// TwinCAT 3 PLC project TcoIoBeckhoff
// Title: TcoIoBeckhoff
// Company: Vortex.Library
// ProjectVersion: 1.19.1.1780
// ProgramVersion: 3.1.4023.0
// libraries:
//   Tc2_EtherCAT, * (Beckhoff Automation GmbH)
//   Tc2_Standard, * (Beckhoff Automation GmbH)
//   Tc2_System, * (Beckhoff Automation GmbH)
//   Tc3_Module, * (Beckhoff Automation GmbH)
//   TcoCore, 1.19.1.1780 (Vortex.Library)
// project tree:
//   Diagnostics/EtherCAT/MasterDevice/ InfoData_E68C61CD.TcDUT (not stored), Inputs_A65FACA4.TcDUT (not stored), Outputs_23C0ED1D.TcDUT (not stored), TcoEthercatDiagnosticsTask.TcPOU, TcoEthercatMasterDeviceState.TcDUT (not stored), ITcoEthercatMasterDevice.TcIO (not stored), TcoEthercatMasterDevice.TcPOU
//   Diagnostics/EtherCAT/MasterDevice/Messenger/ DiagnosticsMessenger.TcPOU (not stored), DiagnosticsMessengers.TcPOU (not stored)
//   Diagnostics/EtherCAT/SyncUnit/ SyncUnitTask_2D604ED5.TcDUT (not stored), TcoSyncUnit.TcPOU, InfoData_2A97D6CF.TcDUT (not stored), ITcoSyncUnit.TcIO (not stored), SyncUnitState.TcDUT (not stored), WcState_0B2B16F9.TcDUT (not stored)
//   Diagnostics/EtherCAT/ TcoEthercat.TcGVL (not stored)
//   / PlcTask.TcTTO (not stored)
//   POUs/ MAIN.TcPOU
// real-time tasks:
//   TASK PlcTask: cycle T#10ms, priority 20, ADS port 350
//   TASK PlcTask1: cycle T#10ms, priority 21, ADS port 351
//   TASK PlcTask2: cycle T#10ms, priority 22, ADS port 352
// I/O:
//   DEVICE Device 1 (EtherCAT), AmsNetId 172.20.10.104.2.1
//     Term 1 (EK1200) [EK1200-5000 EtherCAT Power supply (2A E-Bus)]
//       Term 2 (EL6002) [EL6002 Interface 2Ch. (RS232)]
//       Term 3 (EL1809) [EL1809 16Ch. Dig. Input 24V, 3ms]
//       Term 4 (EL2809) [EL2809 16Ch. Dig. Output 24V, 0.5A]
//       Term 5 (EL4004) [EL4004 4Ch. Ana. Output 0-10V, 12bit]
//       Term 6 (EL2809) [EL2809 16Ch. Dig. Output 24V, 0.5A]
//       Term 7 (EL6001) [EL6001 Interface (RS232)]
//       Term 8 (EL9011) [EL9011 End Terminal]
//   DEVICE Device 4 (EtherCAT), AmsNetId 172.20.10.104.5.1
//     Term 9 (EK1100) [EK1100 EtherCAT Coupler (2A E-Bus)]
//       Term 10 (EL6001) [EL6001 Interface (RS232)]
//       Term 11 (EL1809) [EL1809 16Ch. Dig. Input 24V, 3ms]
//       Term 12 (EL2809) [EL2809 16Ch. Dig. Output 24V, 0.5A]
//       Term 13 (EK1110) [EK1110 EtherCAT extension]
//     Term 14 (EK1100) [EK1100 EtherCAT Coupler (2A E-Bus)]
//       Term 15 (EL3403) [EL3403 3Ch. Power Measuring]
//       Term 16 (EK1122) [EK1122 2 port EtherCAT junction]
//         Term 17 (EK1100) [EK1100 EtherCAT Coupler (2A E-Bus)]
//           Term 18 (EL3174-0002) [EL3174-0002 4Ch. Ana. Input +/-10V, +/-20mA 16 Bit, Isolated Channels]
//           Term 19 (EL6001) [EL6001 Interface (RS232)]
//           Term 20 (EL3011) [EL3011 4Ch. Ana. Input 0-20mA DIFF]
//           Term 21 (EL2008) [EL2008 8Ch. Dig. Output 24V, 0.5A]
//           Term 22 (EL2008) [EL2008 8Ch. Dig. Output 24V, 0.5A]
//           Term 16 (EL9011) [EL9011 End Terminal]
//       Term 23 (EL3024) [EL3024 4Ch. Ana. Input 4-20mA DIFF]
//       Term 17 (EL9011) [EL9011 End Terminal]
// variable links:
//   TcoIoBeckhoffTests/TcoIoBeckhoffTests Instance <-> Device 1 (EtherCAT)
//     PlcTask Inputs/GVL_iXlinker.Device_1_EtherCAT.InfoData.AmsNetId <-> InfoData/AmsNetId
//     PlcTask Inputs/GVL_iXlinker.Device_1_EtherCAT.InfoData.CfgSlaveCount <-> InfoData/CfgSlaveCount
//     PlcTask Inputs/GVL_iXlinker.Device_1_EtherCAT.InfoData.ChangeCount <-> InfoData/ChangeCount
//     PlcTask Inputs/GVL_iXlinker.Device_1_EtherCAT.InfoData.DcToExtTimeOffset <-> InfoData/DcToExtTimeOffset
//     PlcTask Inputs/GVL_iXlinker.Device_1_EtherCAT.InfoData.DcToTcTimeOffset <-> InfoData/DcToTcTimeOffset
//     PlcTask Inputs/GVL_iXlinker.Device_1_EtherCAT.InfoData.DevId <-> InfoData/DevId
//     PlcTask Inputs/GVL_iXlinker.Device_1_EtherCAT.Inputs.DevState <-> Inputs/DevState
//     PlcTask Inputs/GVL_iXlinker.Device_1_EtherCAT.Inputs.Frm0InputToggle <-> Inputs/Frm0InputToggle
//     PlcTask Inputs/GVL_iXlinker.Device_1_EtherCAT.Inputs.Frm0State <-> Inputs/Frm0State
//     PlcTask Inputs/GVL_iXlinker.Device_1_EtherCAT.Inputs.Frm0WcState <-> Inputs/Frm0WcState
//     PlcTask Inputs/GVL_iXlinker.Device_1_EtherCAT.Inputs.SlaveCount <-> Inputs/SlaveCount
//     PlcTask Inputs/GVL_iXlinker.Device_1_EtherCAT.SyncUnits._default.PlcTask1.InfoData.ObjectId <-> SyncUnits/<default>/PlcTask1/InfoData/ObjectId
//     PlcTask Inputs/GVL_iXlinker.Device_1_EtherCAT.SyncUnits._default.PlcTask1.InfoData.SlaveCount <-> SyncUnits/<default>/PlcTask1/InfoData/SlaveCount
//     PlcTask Inputs/GVL_iXlinker.Device_1_EtherCAT.SyncUnits._default.PlcTask1.InfoData.State <-> SyncUnits/<default>/PlcTask1/InfoData/State
//     PlcTask Inputs/GVL_iXlinker.Device_1_EtherCAT.SyncUnits._default.PlcTask1.WcState.WcState <-> SyncUnits/<default>/PlcTask1/WcState/WcState
//     PlcTask Outputs/GVL_iXlinker.Device_1_EtherCAT.Outputs.DevCtrl <-> Outputs/DevCtrl
//     PlcTask Outputs/GVL_iXlinker.Device_1_EtherCAT.Outputs.Frm0Ctrl <-> Outputs/Frm0Ctrl
//     PlcTask Outputs/GVL_iXlinker.Device_1_EtherCAT.Outputs.Frm0WcCtrl <-> Outputs/Frm0WcCtrl
//   TcoIoBeckhoffTests/TcoIoBeckhoffTests Instance <-> Device 1 (EtherCAT)/Term 1 (EK1200)/Term 2 (EL6002)
//     PlcTask Inputs/GVL_iXlinker.Device_1_EtherCAT.Term_1_EK1200.Term_2_EL6002.COM_TxPDO_Map_Inputs_Channel_1.Data_In[0] <-> COM TxPDO-Map Inputs Channel 1/Data In 0
//     PlcTask Inputs/GVL_iXlinker.Device_1_EtherCAT.Term_1_EK1200.Term_2_EL6002.COM_TxPDO_Map_Inputs_Channel_1.Data_In[10] <-> COM TxPDO-Map Inputs Channel 1/Data In 10
//     PlcTask Inputs/GVL_iXlinker.Device_1_EtherCAT.Term_1_EK1200.Term_2_EL6002.COM_TxPDO_Map_Inputs_Channel_1.Data_In[11] <-> COM TxPDO-Map Inputs Channel 1/Data In 11
//     PlcTask Inputs/GVL_iXlinker.Device_1_EtherCAT.Term_1_EK1200.Term_2_EL6002.COM_TxPDO_Map_Inputs_Channel_1.Data_In[12] <-> COM TxPDO-Map Inputs Channel 1/Data In 12
//     PlcTask Inputs/GVL_iXlinker.Device_1_EtherCAT.Term_1_EK1200.Term_2_EL6002.COM_TxPDO_Map_Inputs_Channel_1.Data_In[13] <-> COM TxPDO-Map Inputs Channel 1/Data In 13
//     PlcTask Inputs/GVL_iXlinker.Device_1_EtherCAT.Term_1_EK1200.Term_2_EL6002.COM_TxPDO_Map_Inputs_Channel_1.Data_In[14] <-> COM TxPDO-Map Inputs Channel 1/Data In 14
//     PlcTask Inputs/GVL_iXlinker.Device_1_EtherCAT.Term_1_EK1200.Term_2_EL6002.COM_TxPDO_Map_Inputs_Channel_1.Data_In[15] <-> COM TxPDO-Map Inputs Channel 1/Data In 15
//     PlcTask Inputs/GVL_iXlinker.Device_1_EtherCAT.Term_1_EK1200.Term_2_EL6002.COM_TxPDO_Map_Inputs_Channel_1.Data_In[16] <-> COM TxPDO-Map Inputs Channel 1/Data In 16
//     PlcTask Inputs/GVL_iXlinker.Device_1_EtherCAT.Term_1_EK1200.Term_2_EL6002.COM_TxPDO_Map_Inputs_Channel_1.Data_In[17] <-> COM TxPDO-Map Inputs Channel 1/Data In 17
//     PlcTask Inputs/GVL_iXlinker.Device_1_EtherCAT.Term_1_EK1200.Term_2_EL6002.COM_TxPDO_Map_Inputs_Channel_1.Data_In[18] <-> COM TxPDO-Map Inputs Channel 1/Data In 18
//     PlcTask Inputs/GVL_iXlinker.Device_1_EtherCAT.Term_1_EK1200.Term_2_EL6002.COM_TxPDO_Map_Inputs_Channel_1.Data_In[19] <-> COM TxPDO-Map Inputs Channel 1/Data In 19
//     PlcTask Inputs/GVL_iXlinker.Device_1_EtherCAT.Term_1_EK1200.Term_2_EL6002.COM_TxPDO_Map_Inputs_Channel_1.Data_In[1] <-> COM TxPDO-Map Inputs Channel 1/Data In 1
//     PlcTask Inputs/GVL_iXlinker.Device_1_EtherCAT.Term_1_EK1200.Term_2_EL6002.COM_TxPDO_Map_Inputs_Channel_1.Data_In[20] <-> COM TxPDO-Map Inputs Channel 1/Data In 20
//     PlcTask Inputs/GVL_iXlinker.Device_1_EtherCAT.Term_1_EK1200.Term_2_EL6002.COM_TxPDO_Map_Inputs_Channel_1.Data_In[21] <-> COM TxPDO-Map Inputs Channel 1/Data In 21
//     PlcTask Inputs/GVL_iXlinker.Device_1_EtherCAT.Term_1_EK1200.Term_2_EL6002.COM_TxPDO_Map_Inputs_Channel_1.Data_In[2] <-> COM TxPDO-Map Inputs Channel 1/Data In 2
//     PlcTask Inputs/GVL_iXlinker.Device_1_EtherCAT.Term_1_EK1200.Term_2_EL6002.COM_TxPDO_Map_Inputs_Channel_1.Data_In[3] <-> COM TxPDO-Map Inputs Channel 1/Data In 3
//     PlcTask Inputs/GVL_iXlinker.Device_1_EtherCAT.Term_1_EK1200.Term_2_EL6002.COM_TxPDO_Map_Inputs_Channel_1.Data_In[4] <-> COM TxPDO-Map Inputs Channel 1/Data In 4
//     PlcTask Inputs/GVL_iXlinker.Device_1_EtherCAT.Term_1_EK1200.Term_2_EL6002.COM_TxPDO_Map_Inputs_Channel_1.Data_In[5] <-> COM TxPDO-Map Inputs Channel 1/Data In 5
//     PlcTask Inputs/GVL_iXlinker.Device_1_EtherCAT.Term_1_EK1200.Term_2_EL6002.COM_TxPDO_Map_Inputs_Channel_1.Data_In[6] <-> COM TxPDO-Map Inputs Channel 1/Data In 6
//     PlcTask Inputs/GVL_iXlinker.Device_1_EtherCAT.Term_1_EK1200.Term_2_EL6002.COM_TxPDO_Map_Inputs_Channel_1.Data_In[7] <-> COM TxPDO-Map Inputs Channel 1/Data In 7
//     PlcTask Inputs/GVL_iXlinker.Device_1_EtherCAT.Term_1_EK1200.Term_2_EL6002.COM_TxPDO_Map_Inputs_Channel_1.Data_In[8] <-> COM TxPDO-Map Inputs Channel 1/Data In 8
//     PlcTask Inputs/GVL_iXlinker.Device_1_EtherCAT.Term_1_EK1200.Term_2_EL6002.COM_TxPDO_Map_Inputs_Channel_1.Data_In[9] <-> COM TxPDO-Map Inputs Channel 1/Data In 9
//     PlcTask Inputs/GVL_iXlinker.Device_1_EtherCAT.Term_1_EK1200.Term_2_EL6002.COM_TxPDO_Map_Inputs_Channel_2.Data_In[0] <-> COM TxPDO-Map Inputs Channel 2/Data In 0
//     PlcTask Inputs/GVL_iXlinker.Device_1_EtherCAT.Term_1_EK1200.Term_2_EL6002.COM_TxPDO_Map_Inputs_Channel_2.Data_In[10] <-> COM TxPDO-Map Inputs Channel 2/Data In 10
//     PlcTask Inputs/GVL_iXlinker.Device_1_EtherCAT.Term_1_EK1200.Term_2_EL6002.COM_TxPDO_Map_Inputs_Channel_2.Data_In[11] <-> COM TxPDO-Map Inputs Channel 2/Data In 11
//     PlcTask Inputs/GVL_iXlinker.Device_1_EtherCAT.Term_1_EK1200.Term_2_EL6002.COM_TxPDO_Map_Inputs_Channel_2.Data_In[12] <-> COM TxPDO-Map Inputs Channel 2/Data In 12
//     PlcTask Inputs/GVL_iXlinker.Device_1_EtherCAT.Term_1_EK1200.Term_2_EL6002.COM_TxPDO_Map_Inputs_Channel_2.Data_In[13] <-> COM TxPDO-Map Inputs Channel 2/Data In 13
//     PlcTask Inputs/GVL_iXlinker.Device_1_EtherCAT.Term_1_EK1200.Term_2_EL6002.COM_TxPDO_Map_Inputs_Channel_2.Data_In[14] <-> COM TxPDO-Map Inputs Channel 2/Data In 14
//     PlcTask Inputs/GVL_iXlinker.Device_1_EtherCAT.Term_1_EK1200.Term_2_EL6002.COM_TxPDO_Map_Inputs_Channel_2.Data_In[15] <-> COM TxPDO-Map Inputs Channel 2/Data In 15
//     PlcTask Inputs/GVL_iXlinker.Device_1_EtherCAT.Term_1_EK1200.Term_2_EL6002.COM_TxPDO_Map_Inputs_Channel_2.Data_In[16] <-> COM TxPDO-Map Inputs Channel 2/Data In 16
//     PlcTask Inputs/GVL_iXlinker.Device_1_EtherCAT.Term_1_EK1200.Term_2_EL6002.COM_TxPDO_Map_Inputs_Channel_2.Data_In[17] <-> COM TxPDO-Map Inputs Channel 2/Data In 17
//     PlcTask Inputs/GVL_iXlinker.Device_1_EtherCAT.Term_1_EK1200.Term_2_EL6002.COM_TxPDO_Map_Inputs_Channel_2.Data_In[18] <-> COM TxPDO-Map Inputs Channel 2/Data In 18
//     PlcTask Inputs/GVL_iXlinker.Device_1_EtherCAT.Term_1_EK1200.Term_2_EL6002.COM_TxPDO_Map_Inputs_Channel_2.Data_In[19] <-> COM TxPDO-Map Inputs Channel 2/Data In 19
//     PlcTask Inputs/GVL_iXlinker.Device_1_EtherCAT.Term_1_EK1200.Term_2_EL6002.COM_TxPDO_Map_Inputs_Channel_2.Data_In[1] <-> COM TxPDO-Map Inputs Channel 2/Data In 1
//     PlcTask Inputs/GVL_iXlinker.Device_1_EtherCAT.Term_1_EK1200.Term_2_EL6002.COM_TxPDO_Map_Inputs_Channel_2.Data_In[20] <-> COM TxPDO-Map Inputs Channel 2/Data In 20
//     PlcTask Inputs/GVL_iXlinker.Device_1_EtherCAT.Term_1_EK1200.Term_2_EL6002.COM_TxPDO_Map_Inputs_Channel_2.Data_In[21] <-> COM TxPDO-Map Inputs Channel 2/Data In 21
//     PlcTask Inputs/GVL_iXlinker.Device_1_EtherCAT.Term_1_EK1200.Term_2_EL6002.COM_TxPDO_Map_Inputs_Channel_2.Data_In[2] <-> COM TxPDO-Map Inputs Channel 2/Data In 2
//     PlcTask Inputs/GVL_iXlinker.Device_1_EtherCAT.Term_1_EK1200.Term_2_EL6002.COM_TxPDO_Map_Inputs_Channel_2.Data_In[3] <-> COM TxPDO-Map Inputs Channel 2/Data In 3
//     PlcTask Inputs/GVL_iXlinker.Device_1_EtherCAT.Term_1_EK1200.Term_2_EL6002.COM_TxPDO_Map_Inputs_Channel_2.Data_In[4] <-> COM TxPDO-Map Inputs Channel 2/Data In 4
//     PlcTask Inputs/GVL_iXlinker.Device_1_EtherCAT.Term_1_EK1200.Term_2_EL6002.COM_TxPDO_Map_Inputs_Channel_2.Data_In[5] <-> COM TxPDO-Map Inputs Channel 2/Data In 5
//     PlcTask Inputs/GVL_iXlinker.Device_1_EtherCAT.Term_1_EK1200.Term_2_EL6002.COM_TxPDO_Map_Inputs_Channel_2.Data_In[6] <-> COM TxPDO-Map Inputs Channel 2/Data In 6
//     PlcTask Inputs/GVL_iXlinker.Device_1_EtherCAT.Term_1_EK1200.Term_2_EL6002.COM_TxPDO_Map_Inputs_Channel_2.Data_In[7] <-> COM TxPDO-Map Inputs Channel 2/Data In 7
//     PlcTask Inputs/GVL_iXlinker.Device_1_EtherCAT.Term_1_EK1200.Term_2_EL6002.COM_TxPDO_Map_Inputs_Channel_2.Data_In[8] <-> COM TxPDO-Map Inputs Channel 2/Data In 8
//     PlcTask Inputs/GVL_iXlinker.Device_1_EtherCAT.Term_1_EK1200.Term_2_EL6002.COM_TxPDO_Map_Inputs_Channel_2.Data_In[9] <-> COM TxPDO-Map Inputs Channel 2/Data In 9
//     PlcTask Inputs/GVL_iXlinker.Device_1_EtherCAT.Term_1_EK1200.Term_2_EL6002.COM_TxPDO_Map_Inputs_Channel_1.Status/Buffer_full <-> COM TxPDO-Map Inputs Channel 1/Status/Buffer full
//     PlcTask Inputs/GVL_iXlinker.Device_1_EtherCAT.Term_1_EK1200.Term_2_EL6002.COM_TxPDO_Map_Inputs_Channel_2.Status/Buffer_full <-> COM TxPDO-Map Inputs Channel 2/Status/Buffer full
//     PlcTask Inputs/GVL_iXlinker.Device_1_EtherCAT.Term_1_EK1200.Term_2_EL6002.COM_TxPDO_Map_Inputs_Channel_1.Status/Framing_error <-> COM TxPDO-Map Inputs Channel 1/Status/Framing error
//     PlcTask Inputs/GVL_iXlinker.Device_1_EtherCAT.Term_1_EK1200.Term_2_EL6002.COM_TxPDO_Map_Inputs_Channel_2.Status/Framing_error <-> COM TxPDO-Map Inputs Channel 2/Status/Framing error
//     PlcTask Inputs/GVL_iXlinker.Device_1_EtherCAT.Term_1_EK1200.Term_2_EL6002.COM_TxPDO_Map_Inputs_Channel_1.Status/Init_accepted <-> COM TxPDO-Map Inputs Channel 1/Status/Init accepted
//     PlcTask Inputs/GVL_iXlinker.Device_1_EtherCAT.Term_1_EK1200.Term_2_EL6002.COM_TxPDO_Map_Inputs_Channel_2.Status/Init_accepted <-> COM TxPDO-Map Inputs Channel 2/Status/Init accepted
//     PlcTask Inputs/GVL_iXlinker.Device_1_EtherCAT.Term_1_EK1200.Term_2_EL6002.COM_TxPDO_Map_Inputs_Channel_1.Status/Input_length <-> COM TxPDO-Map Inputs Channel 1/Status/Input length
//     PlcTask Inputs/GVL_iXlinker.Device_1_EtherCAT.Term_1_EK1200.Term_2_EL6002.COM_TxPDO_Map_Inputs_Channel_2.Status/Input_length <-> COM TxPDO-Map Inputs Channel 2/Status/Input length
//     PlcTask Inputs/GVL_iXlinker.Device_1_EtherCAT.Term_1_EK1200.Term_2_EL6002.COM_TxPDO_Map_Inputs_Channel_1.Status/Overrun_error <-> COM TxPDO-Map Inputs Channel 1/Status/Overrun error
//     PlcTask Inputs/GVL_iXlinker.Device_1_EtherCAT.Term_1_EK1200.Term_2_EL6002.COM_TxPDO_Map_Inputs_Channel_2.Status/Overrun_error <-> COM TxPDO-Map Inputs Channel 2/Status/Overrun error
//     PlcTask Inputs/GVL_iXlinker.Device_1_EtherCAT.Term_1_EK1200.Term_2_EL6002.COM_TxPDO_Map_Inputs_Channel_1.Status/Parity_error <-> COM TxPDO-Map Inputs Channel 1/Status/Parity error
//     PlcTask Inputs/GVL_iXlinker.Device_1_EtherCAT.Term_1_EK1200.Term_2_EL6002.COM_TxPDO_Map_Inputs_Channel_2.Status/Parity_error <-> COM TxPDO-Map Inputs Channel 2/Status/Parity error
//     PlcTask Inputs/GVL_iXlinker.Device_1_EtherCAT.Term_1_EK1200.Term_2_EL6002.COM_TxPDO_Map_Inputs_Channel_1.Status/Receive_request <-> COM TxPDO-Map Inputs Channel 1/Status/Receive request
//     PlcTask Inputs/GVL_iXlinker.Device_1_EtherCAT.Term_1_EK1200.Term_2_EL6002.COM_TxPDO_Map_Inputs_Channel_2.Status/Receive_request <-> COM TxPDO-Map Inputs Channel 2/Status/Receive request
//     PlcTask Inputs/GVL_iXlinker.Device_1_EtherCAT.Term_1_EK1200.Term_2_EL6002.COM_TxPDO_Map_Inputs_Channel_1.Status/Transmit_accepted <-> COM TxPDO-Map Inputs Channel 1/Status/Transmit accepted
//     PlcTask Inputs/GVL_iXlinker.Device_1_EtherCAT.Term_1_EK1200.Term_2_EL6002.COM_TxPDO_Map_Inputs_Channel_2.Status/Transmit_accepted <-> COM TxPDO-Map Inputs Channel 2/Status/Transmit accepted
//     PlcTask Inputs/GVL_iXlinker.Device_1_EtherCAT.Term_1_EK1200.Term_2_EL6002.InfoData.AdsAddr <-> InfoData/AdsAddr
//     PlcTask Inputs/GVL_iXlinker.Device_1_EtherCAT.Term_1_EK1200.Term_2_EL6002.InfoData.ObjectId <-> InfoData/ObjectId
//     PlcTask Inputs/GVL_iXlinker.Device_1_EtherCAT.Term_1_EK1200.Term_2_EL6002.InfoData.State <-> InfoData/State
//     PlcTask Inputs/GVL_iXlinker.Device_1_EtherCAT.Term_1_EK1200.Term_2_EL6002.WcState.InputToggle <-> WcState/InputToggle
//     PlcTask Inputs/GVL_iXlinker.Device_1_EtherCAT.Term_1_EK1200.Term_2_EL6002.WcState.WcState <-> WcState/WcState
//     PlcTask Outputs/GVL_iXlinker.Device_1_EtherCAT.Term_1_EK1200.Term_2_EL6002.COM_RxPDO_Map_Outputs_Channel_1.Ctrl/Init_request <-> COM RxPDO-Map Outputs Channel 1/Ctrl/Init request
//     PlcTask Outputs/GVL_iXlinker.Device_1_EtherCAT.Term_1_EK1200.Term_2_EL6002.COM_RxPDO_Map_Outputs_Channel_2.Ctrl/Init_request <-> COM RxPDO-Map Outputs Channel 2/Ctrl/Init request
//     PlcTask Outputs/GVL_iXlinker.Device_1_EtherCAT.Term_1_EK1200.Term_2_EL6002.COM_RxPDO_Map_Outputs_Channel_1.Ctrl/Output_length <-> COM RxPDO-Map Outputs Channel 1/Ctrl/Output length
//     PlcTask Outputs/GVL_iXlinker.Device_1_EtherCAT.Term_1_EK1200.Term_2_EL6002.COM_RxPDO_Map_Outputs_Channel_2.Ctrl/Output_length <-> COM RxPDO-Map Outputs Channel 2/Ctrl/Output length
//     PlcTask Outputs/GVL_iXlinker.Device_1_EtherCAT.Term_1_EK1200.Term_2_EL6002.COM_RxPDO_Map_Outputs_Channel_1.Ctrl/Receive_accepted <-> COM RxPDO-Map Outputs Channel 1/Ctrl/Receive accepted
//     PlcTask Outputs/GVL_iXlinker.Device_1_EtherCAT.Term_1_EK1200.Term_2_EL6002.COM_RxPDO_Map_Outputs_Channel_2.Ctrl/Receive_accepted <-> COM RxPDO-Map Outputs Channel 2/Ctrl/Receive accepted
//     PlcTask Outputs/GVL_iXlinker.Device_1_EtherCAT.Term_1_EK1200.Term_2_EL6002.COM_RxPDO_Map_Outputs_Channel_1.Ctrl/Send_continuous <-> COM RxPDO-Map Outputs Channel 1/Ctrl/Send continuous
//     PlcTask Outputs/GVL_iXlinker.Device_1_EtherCAT.Term_1_EK1200.Term_2_EL6002.COM_RxPDO_Map_Outputs_Channel_2.Ctrl/Send_continuous <-> COM RxPDO-Map Outputs Channel 2/Ctrl/Send continuous
//     PlcTask Outputs/GVL_iXlinker.Device_1_EtherCAT.Term_1_EK1200.Term_2_EL6002.COM_RxPDO_Map_Outputs_Channel_1.Ctrl/Transmit_request <-> COM RxPDO-Map Outputs Channel 1/Ctrl/Transmit request
//     PlcTask Outputs/GVL_iXlinker.Device_1_EtherCAT.Term_1_EK1200.Term_2_EL6002.COM_RxPDO_Map_Outputs_Channel_2.Ctrl/Transmit_request <-> COM RxPDO-Map Outputs Channel 2/Ctrl/Transmit request
//     PlcTask Outputs/GVL_iXlinker.Device_1_EtherCAT.Term_1_EK1200.Term_2_EL6002.COM_RxPDO_Map_Outputs_Channel_1.Data_Out[0] <-> COM RxPDO-Map Outputs Channel 1/Data Out 0
//     PlcTask Outputs/GVL_iXlinker.Device_1_EtherCAT.Term_1_EK1200.Term_2_EL6002.COM_RxPDO_Map_Outputs_Channel_1.Data_Out[10] <-> COM RxPDO-Map Outputs Channel 1/Data Out 10
//     PlcTask Outputs/GVL_iXlinker.Device_1_EtherCAT.Term_1_EK1200.Term_2_EL6002.COM_RxPDO_Map_Outputs_Channel_1.Data_Out[11] <-> COM RxPDO-Map Outputs Channel 1/Data Out 11
//     PlcTask Outputs/GVL_iXlinker.Device_1_EtherCAT.Term_1_EK1200.Term_2_EL6002.COM_RxPDO_Map_Outputs_Channel_1.Data_Out[12] <-> COM RxPDO-Map Outputs Channel 1/Data Out 12
//     PlcTask Outputs/GVL_iXlinker.Device_1_EtherCAT.Term_1_EK1200.Term_2_EL6002.COM_RxPDO_Map_Outputs_Channel_1.Data_Out[13] <-> COM RxPDO-Map Outputs Channel 1/Data Out 13
//     PlcTask Outputs/GVL_iXlinker.Device_1_EtherCAT.Term_1_EK1200.Term_2_EL6002.COM_RxPDO_Map_Outputs_Channel_1.Data_Out[14] <-> COM RxPDO-Map Outputs Channel 1/Data Out 14
//     PlcTask Outputs/GVL_iXlinker.Device_1_EtherCAT.Term_1_EK1200.Term_2_EL6002.COM_RxPDO_Map_Outputs_Channel_1.Data_Out[15] <-> COM RxPDO-Map Outputs Channel 1/Data Out 15
//     PlcTask Outputs/GVL_iXlinker.Device_1_EtherCAT.Term_1_EK1200.Term_2_EL6002.COM_RxPDO_Map_Outputs_Channel_1.Data_Out[16] <-> COM RxPDO-Map Outputs Channel 1/Data Out 16
//     PlcTask Outputs/GVL_iXlinker.Device_1_EtherCAT.Term_1_EK1200.Term_2_EL6002.COM_RxPDO_Map_Outputs_Channel_1.Data_Out[17] <-> COM RxPDO-Map Outputs Channel 1/Data Out 17
//     PlcTask Outputs/GVL_iXlinker.Device_1_EtherCAT.Term_1_EK1200.Term_2_EL6002.COM_RxPDO_Map_Outputs_Channel_1.Data_Out[18] <-> COM RxPDO-Map Outputs Channel 1/Data Out 18
//     PlcTask Outputs/GVL_iXlinker.Device_1_EtherCAT.Term_1_EK1200.Term_2_EL6002.COM_RxPDO_Map_Outputs_Channel_1.Data_Out[19] <-> COM RxPDO-Map Outputs Channel 1/Data Out 19
//     PlcTask Outputs/GVL_iXlinker.Device_1_EtherCAT.Term_1_EK1200.Term_2_EL6002.COM_RxPDO_Map_Outputs_Channel_1.Data_Out[1] <-> COM RxPDO-Map Outputs Channel 1/Data Out 1
//     PlcTask Outputs/GVL_iXlinker.Device_1_EtherCAT.Term_1_EK1200.Term_2_EL6002.COM_RxPDO_Map_Outputs_Channel_1.Data_Out[20] <-> COM RxPDO-Map Outputs Channel 1/Data Out 20
//     PlcTask Outputs/GVL_iXlinker.Device_1_EtherCAT.Term_1_EK1200.Term_2_EL6002.COM_RxPDO_Map_Outputs_Channel_1.Data_Out[21] <-> COM RxPDO-Map Outputs Channel 1/Data Out 21
//     PlcTask Outputs/GVL_iXlinker.Device_1_EtherCAT.Term_1_EK1200.Term_2_EL6002.COM_RxPDO_Map_Outputs_Channel_1.Data_Out[2] <-> COM RxPDO-Map Outputs Channel 1/Data Out 2
//     PlcTask Outputs/GVL_iXlinker.Device_1_EtherCAT.Term_1_EK1200.Term_2_EL6002.COM_RxPDO_Map_Outputs_Channel_1.Data_Out[3] <-> COM RxPDO-Map Outputs Channel 1/Data Out 3
//     PlcTask Outputs/GVL_iXlinker.Device_1_EtherCAT.Term_1_EK1200.Term_2_EL6002.COM_RxPDO_Map_Outputs_Channel_1.Data_Out[4] <-> COM RxPDO-Map Outputs Channel 1/Data Out 4
//     PlcTask Outputs/GVL_iXlinker.Device_1_EtherCAT.Term_1_EK1200.Term_2_EL6002.COM_RxPDO_Map_Outputs_Channel_1.Data_Out[5] <-> COM RxPDO-Map Outputs Channel 1/Data Out 5
//     PlcTask Outputs/GVL_iXlinker.Device_1_EtherCAT.Term_1_EK1200.Term_2_EL6002.COM_RxPDO_Map_Outputs_Channel_1.Data_Out[6] <-> COM RxPDO-Map Outputs Channel 1/Data Out 6
//     PlcTask Outputs/GVL_iXlinker.Device_1_EtherCAT.Term_1_EK1200.Term_2_EL6002.COM_RxPDO_Map_Outputs_Channel_1.Data_Out[7] <-> COM RxPDO-Map Outputs Channel 1/Data Out 7
//     PlcTask Outputs/GVL_iXlinker.Device_1_EtherCAT.Term_1_EK1200.Term_2_EL6002.COM_RxPDO_Map_Outputs_Channel_1.Data_Out[8] <-> COM RxPDO-Map Outputs Channel 1/Data Out 8
//     PlcTask Outputs/GVL_iXlinker.Device_1_EtherCAT.Term_1_EK1200.Term_2_EL6002.COM_RxPDO_Map_Outputs_Channel_1.Data_Out[9] <-> COM RxPDO-Map Outputs Channel 1/Data Out 9
//     PlcTask Outputs/GVL_iXlinker.Device_1_EtherCAT.Term_1_EK1200.Term_2_EL6002.COM_RxPDO_Map_Outputs_Channel_2.Data_Out[0] <-> COM RxPDO-Map Outputs Channel 2/Data Out 0
//     PlcTask Outputs/GVL_iXlinker.Device_1_EtherCAT.Term_1_EK1200.Term_2_EL6002.COM_RxPDO_Map_Outputs_Channel_2.Data_Out[10] <-> COM RxPDO-Map Outputs Channel 2/Data Out 10
//     PlcTask Outputs/GVL_iXlinker.Device_1_EtherCAT.Term_1_EK1200.Term_2_EL6002.COM_RxPDO_Map_Outputs_Channel_2.Data_Out[11] <-> COM RxPDO-Map Outputs Channel 2/Data Out 11
//     PlcTask Outputs/GVL_iXlinker.Device_1_EtherCAT.Term_1_EK1200.Term_2_EL6002.COM_RxPDO_Map_Outputs_Channel_2.Data_Out[12] <-> COM RxPDO-Map Outputs Channel 2/Data Out 12
//     PlcTask Outputs/GVL_iXlinker.Device_1_EtherCAT.Term_1_EK1200.Term_2_EL6002.COM_RxPDO_Map_Outputs_Channel_2.Data_Out[13] <-> COM RxPDO-Map Outputs Channel 2/Data Out 13
//     PlcTask Outputs/GVL_iXlinker.Device_1_EtherCAT.Term_1_EK1200.Term_2_EL6002.COM_RxPDO_Map_Outputs_Channel_2.Data_Out[14] <-> COM RxPDO-Map Outputs Channel 2/Data Out 14
//     PlcTask Outputs/GVL_iXlinker.Device_1_EtherCAT.Term_1_EK1200.Term_2_EL6002.COM_RxPDO_Map_Outputs_Channel_2.Data_Out[15] <-> COM RxPDO-Map Outputs Channel 2/Data Out 15
//     PlcTask Outputs/GVL_iXlinker.Device_1_EtherCAT.Term_1_EK1200.Term_2_EL6002.COM_RxPDO_Map_Outputs_Channel_2.Data_Out[16] <-> COM RxPDO-Map Outputs Channel 2/Data Out 16
//     PlcTask Outputs/GVL_iXlinker.Device_1_EtherCAT.Term_1_EK1200.Term_2_EL6002.COM_RxPDO_Map_Outputs_Channel_2.Data_Out[17] <-> COM RxPDO-Map Outputs Channel 2/Data Out 17
//     PlcTask Outputs/GVL_iXlinker.Device_1_EtherCAT.Term_1_EK1200.Term_2_EL6002.COM_RxPDO_Map_Outputs_Channel_2.Data_Out[18] <-> COM RxPDO-Map Outputs Channel 2/Data Out 18
//     PlcTask Outputs/GVL_iXlinker.Device_1_EtherCAT.Term_1_EK1200.Term_2_EL6002.COM_RxPDO_Map_Outputs_Channel_2.Data_Out[19] <-> COM RxPDO-Map Outputs Channel 2/Data Out 19
//     PlcTask Outputs/GVL_iXlinker.Device_1_EtherCAT.Term_1_EK1200.Term_2_EL6002.COM_RxPDO_Map_Outputs_Channel_2.Data_Out[1] <-> COM RxPDO-Map Outputs Channel 2/Data Out 1
//     PlcTask Outputs/GVL_iXlinker.Device_1_EtherCAT.Term_1_EK1200.Term_2_EL6002.COM_RxPDO_Map_Outputs_Channel_2.Data_Out[20] <-> COM RxPDO-Map Outputs Channel 2/Data Out 20
//     PlcTask Outputs/GVL_iXlinker.Device_1_EtherCAT.Term_1_EK1200.Term_2_EL6002.COM_RxPDO_Map_Outputs_Channel_2.Data_Out[21] <-> COM RxPDO-Map Outputs Channel 2/Data Out 21
//     PlcTask Outputs/GVL_iXlinker.Device_1_EtherCAT.Term_1_EK1200.Term_2_EL6002.COM_RxPDO_Map_Outputs_Channel_2.Data_Out[2] <-> COM RxPDO-Map Outputs Channel 2/Data Out 2
//     PlcTask Outputs/GVL_iXlinker.Device_1_EtherCAT.Term_1_EK1200.Term_2_EL6002.COM_RxPDO_Map_Outputs_Channel_2.Data_Out[3] <-> COM RxPDO-Map Outputs Channel 2/Data Out 3
//     PlcTask Outputs/GVL_iXlinker.Device_1_EtherCAT.Term_1_EK1200.Term_2_EL6002.COM_RxPDO_Map_Outputs_Channel_2.Data_Out[4] <-> COM RxPDO-Map Outputs Channel 2/Data Out 4
//     PlcTask Outputs/GVL_iXlinker.Device_1_EtherCAT.Term_1_EK1200.Term_2_EL6002.COM_RxPDO_Map_Outputs_Channel_2.Data_Out[5] <-> COM RxPDO-Map Outputs Channel 2/Data Out 5
//     PlcTask Outputs/GVL_iXlinker.Device_1_EtherCAT.Term_1_EK1200.Term_2_EL6002.COM_RxPDO_Map_Outputs_Channel_2.Data_Out[6] <-> COM RxPDO-Map Outputs Channel 2/Data Out 6
//     PlcTask Outputs/GVL_iXlinker.Device_1_EtherCAT.Term_1_EK1200.Term_2_EL6002.COM_RxPDO_Map_Outputs_Channel_2.Data_Out[7] <-> COM RxPDO-Map Outputs Channel 2/Data Out 7
//     PlcTask Outputs/GVL_iXlinker.Device_1_EtherCAT.Term_1_EK1200.Term_2_EL6002.COM_RxPDO_Map_Outputs_Channel_2.Data_Out[8] <-> COM RxPDO-Map Outputs Channel 2/Data Out 8
//     PlcTask Outputs/GVL_iXlinker.Device_1_EtherCAT.Term_1_EK1200.Term_2_EL6002.COM_RxPDO_Map_Outputs_Channel_2.Data_Out[9] <-> COM RxPDO-Map Outputs Channel 2/Data Out 9
//   TcoIoBeckhoffTests/TcoIoBeckhoffTests Instance <-> Device 1 (EtherCAT)/Term 1 (EK1200)/Term 3 (EL1809)
//     PlcTask Inputs/GVL_iXlinker.Device_1_EtherCAT.Term_1_EK1200.Term_3_EL1809.Channel_{1..16}.Input <-> Channel {1..16}/Input  (16 links)
//     PlcTask Inputs/GVL_iXlinker.Device_1_EtherCAT.Term_1_EK1200.Term_3_EL1809.InfoData.AdsAddr <-> InfoData/AdsAddr
//     PlcTask Inputs/GVL_iXlinker.Device_1_EtherCAT.Term_1_EK1200.Term_3_EL1809.InfoData.ObjectId <-> InfoData/ObjectId
//     PlcTask Inputs/GVL_iXlinker.Device_1_EtherCAT.Term_1_EK1200.Term_3_EL1809.InfoData.State <-> InfoData/State
//     PlcTask Inputs/GVL_iXlinker.Device_1_EtherCAT.Term_1_EK1200.Term_3_EL1809.WcState.InputToggle <-> WcState/InputToggle
//     PlcTask Inputs/GVL_iXlinker.Device_1_EtherCAT.Term_1_EK1200.Term_3_EL1809.WcState.WcState <-> WcState/WcState
//   TcoIoBeckhoffTests/TcoIoBeckhoffTests Instance <-> Device 1 (EtherCAT)/Term 1 (EK1200)/Term 4 (EL2809)
//     PlcTask Inputs/GVL_iXlinker.Device_1_EtherCAT.Term_1_EK1200.Term_4_EL2809.InfoData.AdsAddr <-> InfoData/AdsAddr
//     PlcTask Inputs/GVL_iXlinker.Device_1_EtherCAT.Term_1_EK1200.Term_4_EL2809.InfoData.ObjectId <-> InfoData/ObjectId
//     PlcTask Inputs/GVL_iXlinker.Device_1_EtherCAT.Term_1_EK1200.Term_4_EL2809.InfoData.State <-> InfoData/State
//     PlcTask Inputs/GVL_iXlinker.Device_1_EtherCAT.Term_1_EK1200.Term_4_EL2809.WcState.WcState <-> WcState/WcState
//     PlcTask Outputs/GVL_iXlinker.Device_1_EtherCAT.Term_1_EK1200.Term_4_EL2809.Channel_{1..16}.Output <-> Channel {1..16}/Output  (16 links)
//   TcoIoBeckhoffTests/TcoIoBeckhoffTests Instance <-> Device 1 (EtherCAT)/Term 1 (EK1200)/Term 5 (EL4004)
//     PlcTask Inputs/GVL_iXlinker.Device_1_EtherCAT.Term_1_EK1200.Term_5_EL4004.InfoData.AdsAddr <-> InfoData/AdsAddr
//     PlcTask Inputs/GVL_iXlinker.Device_1_EtherCAT.Term_1_EK1200.Term_5_EL4004.InfoData.ObjectId <-> InfoData/ObjectId
//     PlcTask Inputs/GVL_iXlinker.Device_1_EtherCAT.Term_1_EK1200.Term_5_EL4004.InfoData.State <-> InfoData/State
//     PlcTask Inputs/GVL_iXlinker.Device_1_EtherCAT.Term_1_EK1200.Term_5_EL4004.WcState.WcState <-> WcState/WcState
//     PlcTask Outputs/GVL_iXlinker.Device_1_EtherCAT.Term_1_EK1200.Term_5_EL4004.AO_Outputs_Channel_{1..4}.Analog_output <-> AO Outputs Channel {1..4}/Analog output  (4 links)
//   TcoIoBeckhoffTests/TcoIoBeckhoffTests Instance <-> Device 1 (EtherCAT)/Term 1 (EK1200)/Term 6 (EL2809)
//     PlcTask Inputs/GVL_iXlinker.Device_1_EtherCAT.Term_1_EK1200.Term_6_EL2809.InfoData.AdsAddr <-> InfoData/AdsAddr
//     PlcTask Inputs/GVL_iXlinker.Device_1_EtherCAT.Term_1_EK1200.Term_6_EL2809.InfoData.ObjectId <-> InfoData/ObjectId
//     PlcTask Inputs/GVL_iXlinker.Device_1_EtherCAT.Term_1_EK1200.Term_6_EL2809.InfoData.State <-> InfoData/State
//     PlcTask Inputs/GVL_iXlinker.Device_1_EtherCAT.Term_1_EK1200.Term_6_EL2809.WcState.WcState <-> WcState/WcState
//     PlcTask Outputs/GVL_iXlinker.Device_1_EtherCAT.Term_1_EK1200.Term_6_EL2809.Channel_{1..16}.Output <-> Channel {1..16}/Output  (16 links)
//   TcoIoBeckhoffTests/TcoIoBeckhoffTests Instance <-> Device 1 (EtherCAT)/Term 1 (EK1200)/Term 7 (EL6001)
//     PlcTask Inputs/GVL_iXlinker.Device_1_EtherCAT.Term_1_EK1200.Term_7_EL6001.COM_Inputs.Data_In[{0..21}] <-> COM Inputs/Data In {0..21}  (22 links)
//     PlcTask Inputs/GVL_iXlinker.Device_1_EtherCAT.Term_1_EK1200.Term_7_EL6001.COM_Inputs.Status/Buffer_full <-> COM Inputs/Status/Buffer full
//     PlcTask Inputs/GVL_iXlinker.Device_1_EtherCAT.Term_1_EK1200.Term_7_EL6001.COM_Inputs.Status/Framing_error <-> COM Inputs/Status/Framing error
//     PlcTask Inputs/GVL_iXlinker.Device_1_EtherCAT.Term_1_EK1200.Term_7_EL6001.COM_Inputs.Status/Init_accepted <-> COM Inputs/Status/Init accepted
//     PlcTask Inputs/GVL_iXlinker.Device_1_EtherCAT.Term_1_EK1200.Term_7_EL6001.COM_Inputs.Status/Input_length <-> COM Inputs/Status/Input length
//     PlcTask Inputs/GVL_iXlinker.Device_1_EtherCAT.Term_1_EK1200.Term_7_EL6001.COM_Inputs.Status/Overrun_error <-> COM Inputs/Status/Overrun error
//     PlcTask Inputs/GVL_iXlinker.Device_1_EtherCAT.Term_1_EK1200.Term_7_EL6001.COM_Inputs.Status/Parity_error <-> COM Inputs/Status/Parity error
//     PlcTask Inputs/GVL_iXlinker.Device_1_EtherCAT.Term_1_EK1200.Term_7_EL6001.COM_Inputs.Status/Receive_request <-> COM Inputs/Status/Receive request
//     PlcTask Inputs/GVL_iXlinker.Device_1_EtherCAT.Term_1_EK1200.Term_7_EL6001.COM_Inputs.Status/Transmit_accepted <-> COM Inputs/Status/Transmit accepted
//     PlcTask Inputs/GVL_iXlinker.Device_1_EtherCAT.Term_1_EK1200.Term_7_EL6001.InfoData.AdsAddr <-> InfoData/AdsAddr
//     PlcTask Inputs/GVL_iXlinker.Device_1_EtherCAT.Term_1_EK1200.Term_7_EL6001.InfoData.ObjectId <-> InfoData/ObjectId
//     PlcTask Inputs/GVL_iXlinker.Device_1_EtherCAT.Term_1_EK1200.Term_7_EL6001.InfoData.State <-> InfoData/State
//     PlcTask Inputs/GVL_iXlinker.Device_1_EtherCAT.Term_1_EK1200.Term_7_EL6001.WcState.InputToggle <-> WcState/InputToggle
//     PlcTask Inputs/GVL_iXlinker.Device_1_EtherCAT.Term_1_EK1200.Term_7_EL6001.WcState.WcState <-> WcState/WcState
//     PlcTask Outputs/GVL_iXlinker.Device_1_EtherCAT.Term_1_EK1200.Term_7_EL6001.COM_Outputs.Ctrl/Init_request <-> COM Outputs/Ctrl/Init request
//     PlcTask Outputs/GVL_iXlinker.Device_1_EtherCAT.Term_1_EK1200.Term_7_EL6001.COM_Outputs.Ctrl/Output_length <-> COM Outputs/Ctrl/Output length
//     PlcTask Outputs/GVL_iXlinker.Device_1_EtherCAT.Term_1_EK1200.Term_7_EL6001.COM_Outputs.Ctrl/Receive_accepted <-> COM Outputs/Ctrl/Receive accepted
//     PlcTask Outputs/GVL_iXlinker.Device_1_EtherCAT.Term_1_EK1200.Term_7_EL6001.COM_Outputs.Ctrl/Send_continues <-> COM Outputs/Ctrl/Send continues
//     PlcTask Outputs/GVL_iXlinker.Device_1_EtherCAT.Term_1_EK1200.Term_7_EL6001.COM_Outputs.Ctrl/Transmit_request <-> COM Outputs/Ctrl/Transmit request
//     PlcTask Outputs/GVL_iXlinker.Device_1_EtherCAT.Term_1_EK1200.Term_7_EL6001.COM_Outputs.Data_Out[{0..21}] <-> COM Outputs/Data Out {0..21}  (22 links)
//   TcoIoBeckhoffTests/TcoIoBeckhoffTests Instance <-> Device 4 (EtherCAT)
//     PlcTask Inputs/GVL_iXlinker.Device_4_EtherCAT.InfoData.AmsNetId <-> InfoData/AmsNetId
//     PlcTask Inputs/GVL_iXlinker.Device_4_EtherCAT.InfoData.CfgSlaveCount <-> InfoData/CfgSlaveCount
//     PlcTask Inputs/GVL_iXlinker.Device_4_EtherCAT.InfoData.ChangeCount <-> InfoData/ChangeCount
//     PlcTask Inputs/GVL_iXlinker.Device_4_EtherCAT.InfoData.DcToExtTimeOffset <-> InfoData/DcToExtTimeOffset
//     PlcTask Inputs/GVL_iXlinker.Device_4_EtherCAT.InfoData.DcToTcTimeOffset <-> InfoData/DcToTcTimeOffset
//     PlcTask Inputs/GVL_iXlinker.Device_4_EtherCAT.InfoData.DevId <-> InfoData/DevId
//     PlcTask Inputs/GVL_iXlinker.Device_4_EtherCAT.Inputs.DevState <-> Inputs/DevState
//     PlcTask Inputs/GVL_iXlinker.Device_4_EtherCAT.Inputs.Frm0InputToggle <-> Inputs/Frm0InputToggle
//     PlcTask Inputs/GVL_iXlinker.Device_4_EtherCAT.Inputs.Frm0State <-> Inputs/Frm0State
//     PlcTask Inputs/GVL_iXlinker.Device_4_EtherCAT.Inputs.Frm0WcState <-> Inputs/Frm0WcState
//     PlcTask Inputs/GVL_iXlinker.Device_4_EtherCAT.Inputs.SlaveCount <-> Inputs/SlaveCount
//     PlcTask Inputs/GVL_iXlinker.Device_4_EtherCAT.SyncUnits._default.PlcTask1.InfoData.ObjectId <-> SyncUnits/<default>/PlcTask1/InfoData/ObjectId
//     PlcTask Inputs/GVL_iXlinker.Device_4_EtherCAT.SyncUnits._default.PlcTask1.InfoData.SlaveCount <-> SyncUnits/<default>/PlcTask1/InfoData/SlaveCount
//     PlcTask Inputs/GVL_iXlinker.Device_4_EtherCAT.SyncUnits._default.PlcTask1.InfoData.State <-> SyncUnits/<default>/PlcTask1/InfoData/State
//     PlcTask Inputs/GVL_iXlinker.Device_4_EtherCAT.SyncUnits._default.PlcTask1.WcState.WcState <-> SyncUnits/<default>/PlcTask1/WcState/WcState
//     PlcTask Outputs/GVL_iXlinker.Device_4_EtherCAT.Outputs.DevCtrl <-> Outputs/DevCtrl
//     PlcTask Outputs/GVL_iXlinker.Device_4_EtherCAT.Outputs.Frm0Ctrl <-> Outputs/Frm0Ctrl
//     PlcTask Outputs/GVL_iXlinker.Device_4_EtherCAT.Outputs.Frm0WcCtrl <-> Outputs/Frm0WcCtrl
//   TcoIoBeckhoffTests/TcoIoBeckhoffTests Instance <-> Device 4 (EtherCAT)/Term 14 (EK1100)
//     PlcTask Inputs/GVL_iXlinker.Device_4_EtherCAT.Term_14_EK1100.InfoData.AdsAddr <-> InfoData/AdsAddr
//     PlcTask Inputs/GVL_iXlinker.Device_4_EtherCAT.Term_14_EK1100.InfoData.ObjectId <-> InfoData/ObjectId
//     PlcTask Inputs/GVL_iXlinker.Device_4_EtherCAT.Term_14_EK1100.InfoData.State <-> InfoData/State
//   TcoIoBeckhoffTests/TcoIoBeckhoffTests Instance <-> Device 4 (EtherCAT)/Term 14 (EK1100)/Term 15 (EL3403)
//     PlcTask Inputs/GVL_iXlinker.Device_4_EtherCAT.Term_14_EK1100.Term_15_EL3403.InfoData.AdsAddr <-> InfoData/AdsAddr
//     PlcTask Inputs/GVL_iXlinker.Device_4_EtherCAT.Term_14_EK1100.Term_15_EL3403.InfoData.ObjectId <-> InfoData/ObjectId
//     PlcTask Inputs/GVL_iXlinker.Device_4_EtherCAT.Term_14_EK1100.Term_15_EL3403.InfoData.State <-> InfoData/State
//     PlcTask Inputs/GVL_iXlinker.Device_4_EtherCAT.Term_14_EK1100.Term_15_EL3403.PM_Inputs_Channel_1.Active_power <-> PM Inputs Channel 1/Active power
//     PlcTask Inputs/GVL_iXlinker.Device_4_EtherCAT.Term_14_EK1100.Term_15_EL3403.PM_Inputs_Channel_2.Active_power <-> PM Inputs Channel 2/Active power
//     PlcTask Inputs/GVL_iXlinker.Device_4_EtherCAT.Term_14_EK1100.Term_15_EL3403.PM_Inputs_Channel_3.Active_power <-> PM Inputs Channel 3/Active power
//     PlcTask Inputs/GVL_iXlinker.Device_4_EtherCAT.Term_14_EK1100.Term_15_EL3403.PM_Inputs_Channel_1.Current <-> PM Inputs Channel 1/Current
//     PlcTask Inputs/GVL_iXlinker.Device_4_EtherCAT.Term_14_EK1100.Term_15_EL3403.PM_Inputs_Channel_2.Current <-> PM Inputs Channel 2/Current
//     PlcTask Inputs/GVL_iXlinker.Device_4_EtherCAT.Term_14_EK1100.Term_15_EL3403.PM_Inputs_Channel_3.Current <-> PM Inputs Channel 3/Current
//     PlcTask Inputs/GVL_iXlinker.Device_4_EtherCAT.Term_14_EK1100.Term_15_EL3403.PM_Inputs_Channel_1.Index <-> PM Inputs Channel 1/Index
//     PlcTask Inputs/GVL_iXlinker.Device_4_EtherCAT.Term_14_EK1100.Term_15_EL3403.PM_Inputs_Channel_2.Index <-> PM Inputs Channel 2/Index
//     PlcTask Inputs/GVL_iXlinker.Device_4_EtherCAT.Term_14_EK1100.Term_15_EL3403.PM_Inputs_Channel_3.Index <-> PM Inputs Channel 3/Index
//     PlcTask Inputs/GVL_iXlinker.Device_4_EtherCAT.Term_14_EK1100.Term_15_EL3403.PM_Inputs_Channel_1.TxPDO_Toggle <-> PM Inputs Channel 1/TxPDO Toggle
//     PlcTask Inputs/GVL_iXlinker.Device_4_EtherCAT.Term_14_EK1100.Term_15_EL3403.PM_Inputs_Channel_2.TxPDO_Toggle <-> PM Inputs Channel 2/TxPDO Toggle
//     PlcTask Inputs/GVL_iXlinker.Device_4_EtherCAT.Term_14_EK1100.Term_15_EL3403.PM_Inputs_Channel_3.TxPDO_Toggle <-> PM Inputs Channel 3/TxPDO Toggle
//     PlcTask Inputs/GVL_iXlinker.Device_4_EtherCAT.Term_14_EK1100.Term_15_EL3403.PM_Inputs_Channel_1.Variant_value <-> PM Inputs Channel 1/Variant value
//     PlcTask Inputs/GVL_iXlinker.Device_4_EtherCAT.Term_14_EK1100.Term_15_EL3403.PM_Inputs_Channel_2.Variant_value <-> PM Inputs Channel 2/Variant value
//     PlcTask Inputs/GVL_iXlinker.Device_4_EtherCAT.Term_14_EK1100.Term_15_EL3403.PM_Inputs_Channel_3.Variant_value <-> PM Inputs Channel 3/Variant value
//     PlcTask Inputs/GVL_iXlinker.Device_4_EtherCAT.Term_14_EK1100.Term_15_EL3403.PM_Inputs_Channel_1.Voltage <-> PM Inputs Channel 1/Voltage
//     PlcTask Inputs/GVL_iXlinker.Device_4_EtherCAT.Term_14_EK1100.Term_15_EL3403.PM_Inputs_Channel_2.Voltage <-> PM Inputs Channel 2/Voltage
//     PlcTask Inputs/GVL_iXlinker.Device_4_EtherCAT.Term_14_EK1100.Term_15_EL3403.PM_Inputs_Channel_3.Voltage <-> PM Inputs Channel 3/Voltage
//     PlcTask Inputs/GVL_iXlinker.Device_4_EtherCAT.Term_14_EK1100.Term_15_EL3403.PM_Status_data.Missing_zero_crossing_A <-> PM Status data/Missing zero crossing A
//     PlcTask Inputs/GVL_iXlinker.Device_4_EtherCAT.Term_14_EK1100.Term_15_EL3403.PM_Status_data.Missing_zero_crossing_B <-> PM Status data/Missing zero crossing B
//     PlcTask Inputs/GVL_iXlinker.Device_4_EtherCAT.Term_14_EK1100.Term_15_EL3403.PM_Status_data.Missing_zero_crossing_C <-> PM Status data/Missing zero crossing C
//     PlcTask Inputs/GVL_iXlinker.Device_4_EtherCAT.Term_14_EK1100.Term_15_EL3403.PM_Status_data.Phase_sequence_error <-> PM Status data/Phase sequence error
//     PlcTask Inputs/GVL_iXlinker.Device_4_EtherCAT.Term_14_EK1100.Term_15_EL3403.WcState.InputToggle <-> WcState/InputToggle
//     PlcTask Inputs/GVL_iXlinker.Device_4_EtherCAT.Term_14_EK1100.Term_15_EL3403.WcState.WcState <-> WcState/WcState
//     PlcTask Outputs/GVL_iXlinker.Device_4_EtherCAT.Term_14_EK1100.Term_15_EL3403.PM_Outputs_Channel_1.Index <-> PM Outputs Channel 1/Index
//     PlcTask Outputs/GVL_iXlinker.Device_4_EtherCAT.Term_14_EK1100.Term_15_EL3403.PM_Outputs_Channel_2.Index <-> PM Outputs Channel 2/Index
//     PlcTask Outputs/GVL_iXlinker.Device_4_EtherCAT.Term_14_EK1100.Term_15_EL3403.PM_Outputs_Channel_3.Index <-> PM Outputs Channel 3/Index
//   TcoIoBeckhoffTests/TcoIoBeckhoffTests Instance <-> Device 4 (EtherCAT)/Term 14 (EK1100)/Term 16 (EK1122)
//     PlcTask Inputs/GVL_iXlinker.Device_4_EtherCAT.Term_14_EK1100.Term_16_EK1122.InfoData.AdsAddr <-> InfoData/AdsAddr
//     PlcTask Inputs/GVL_iXlinker.Device_4_EtherCAT.Term_14_EK1100.Term_16_EK1122.InfoData.ObjectId <-> InfoData/ObjectId
//     PlcTask Inputs/GVL_iXlinker.Device_4_EtherCAT.Term_14_EK1100.Term_16_EK1122.InfoData.State <-> InfoData/State
//   TcoIoBeckhoffTests/TcoIoBeckhoffTests Instance <-> Device 4 (EtherCAT)/Term 14 (EK1100)/Term 16 (EK1122)/Term 17 (EK1100)
//     PlcTask Inputs/GVL_iXlinker.Device_4_EtherCAT.Term_14_EK1100.Term_16_EK1122.Term_17_EK1100.InfoData.AdsAddr <-> InfoData/AdsAddr
//     PlcTask Inputs/GVL_iXlinker.Device_4_EtherCAT.Term_14_EK1100.Term_16_EK1122.Term_17_EK1100.InfoData.ObjectId <-> InfoData/ObjectId
//     PlcTask Inputs/GVL_iXlinker.Device_4_EtherCAT.Term_14_EK1100.Term_16_EK1122.Term_17_EK1100.InfoData.State <-> InfoData/State
//   TcoIoBeckhoffTests/TcoIoBeckhoffTests Instance <-> Device 4 (EtherCAT)/Term 14 (EK1100)/Term 16 (EK1122)/Term 17 (EK1100)/Term 18 (EL3174-0002)
//     PlcTask Inputs/GVL_iXlinker.Device_4_EtherCAT.Term_14_EK1100.Term_16_EK1122.Term_17_EK1100.Term_18_EL3174_0002.AI_Standard_Channel_1.Status/Error <-> AI Standard Channel 1/Status/Error
//     PlcTask Inputs/GVL_iXlinker.Device_4_EtherCAT.Term_14_EK1100.Term_16_EK1122.Term_17_EK1100.Term_18_EL3174_0002.AI_Standard_Channel_2.Status/Error <-> AI Standard Channel 2/Status/Error
//     PlcTask Inputs/GVL_iXlinker.Device_4_EtherCAT.Term_14_EK1100.Term_16_EK1122.Term_17_EK1100.Term_18_EL3174_0002.AI_Standard_Channel_3.Status/Error <-> AI Standard Channel 3/Status/Error
//     PlcTask Inputs/GVL_iXlinker.Device_4_EtherCAT.Term_14_EK1100.Term_16_EK1122.Term_17_EK1100.Term_18_EL3174_0002.AI_Standard_Channel_4.Status/Error <-> AI Standard Channel 4/Status/Error
//     PlcTask Inputs/GVL_iXlinker.Device_4_EtherCAT.Term_14_EK1100.Term_16_EK1122.Term_17_EK1100.Term_18_EL3174_0002.AI_Standard_Channel_1.Status/Limit_1 <-> AI Standard Channel 1/Status/Limit 1
//     PlcTask Inputs/GVL_iXlinker.Device_4_EtherCAT.Term_14_EK1100.Term_16_EK1122.Term_17_EK1100.Term_18_EL3174_0002.AI_Standard_Channel_1.Status/Limit_2 <-> AI Standard Channel 1/Status/Limit 2
//     PlcTask Inputs/GVL_iXlinker.Device_4_EtherCAT.Term_14_EK1100.Term_16_EK1122.Term_17_EK1100.Term_18_EL3174_0002.AI_Standard_Channel_2.Status/Limit_1 <-> AI Standard Channel 2/Status/Limit 1
//     PlcTask Inputs/GVL_iXlinker.Device_4_EtherCAT.Term_14_EK1100.Term_16_EK1122.Term_17_EK1100.Term_18_EL3174_0002.AI_Standard_Channel_2.Status/Limit_2 <-> AI Standard Channel 2/Status/Limit 2
//     PlcTask Inputs/GVL_iXlinker.Device_4_EtherCAT.Term_14_EK1100.Term_16_EK1122.Term_17_EK1100.Term_18_EL3174_0002.AI_Standard_Channel_3.Status/Limit_1 <-> AI Standard Channel 3/Status/Limit 1
//     PlcTask Inputs/GVL_iXlinker.Device_4_EtherCAT.Term_14_EK1100.Term_16_EK1122.Term_17_EK1100.Term_18_EL3174_0002.AI_Standard_Channel_3.Status/Limit_2 <-> AI Standard Channel 3/Status/Limit 2
//     PlcTask Inputs/GVL_iXlinker.Device_4_EtherCAT.Term_14_EK1100.Term_16_EK1122.Term_17_EK1100.Term_18_EL3174_0002.AI_Standard_Channel_4.Status/Limit_1 <-> AI Standard Channel 4/Status/Limit 1
//     PlcTask Inputs/GVL_iXlinker.Device_4_EtherCAT.Term_14_EK1100.Term_16_EK1122.Term_17_EK1100.Term_18_EL3174_0002.AI_Standard_Channel_4.Status/Limit_2 <-> AI Standard Channel 4/Status/Limit 2
//     PlcTask Inputs/GVL_iXlinker.Device_4_EtherCAT.Term_14_EK1100.Term_16_EK1122.Term_17_EK1100.Term_18_EL3174_0002.AI_Standard_Channel_1.Status/Overrange <-> AI Standard Channel 1/Status/Overrange
//     PlcTask Inputs/GVL_iXlinker.Device_4_EtherCAT.Term_14_EK1100.Term_16_EK1122.Term_17_EK1100.Term_18_EL3174_0002.AI_Standard_Channel_2.Status/Overrange <-> AI Standard Channel 2/Status/Overrange
//     PlcTask Inputs/GVL_iXlinker.Device_4_EtherCAT.Term_14_EK1100.Term_16_EK1122.Term_17_EK1100.Term_18_EL3174_0002.AI_Standard_Channel_3.Status/Overrange <-> AI Standard Channel 3/Status/Overrange
//     PlcTask Inputs/GVL_iXlinker.Device_4_EtherCAT.Term_14_EK1100.Term_16_EK1122.Term_17_EK1100.Term_18_EL3174_0002.AI_Standard_Channel_4.Status/Overrange <-> AI Standard Channel 4/Status/Overrange
//     PlcTask Inputs/GVL_iXlinker.Device_4_EtherCAT.Term_14_EK1100.Term_16_EK1122.Term_17_EK1100.Term_18_EL3174_0002.AI_Standard_Channel_1.Status/Sync_error <-> AI Standard Channel 1/Status/Sync error
//     PlcTask Inputs/GVL_iXlinker.Device_4_EtherCAT.Term_14_EK1100.Term_16_EK1122.Term_17_EK1100.Term_18_EL3174_0002.AI_Standard_Channel_2.Status/Sync_error <-> AI Standard Channel 2/Status/Sync error
//     PlcTask Inputs/GVL_iXlinker.Device_4_EtherCAT.Term_14_EK1100.Term_16_EK1122.Term_17_EK1100.Term_18_EL3174_0002.AI_Standard_Channel_3.Status/Sync_error <-> AI Standard Channel 3/Status/Sync error
//     PlcTask Inputs/GVL_iXlinker.Device_4_EtherCAT.Term_14_EK1100.Term_16_EK1122.Term_17_EK1100.Term_18_EL3174_0002.AI_Standard_Channel_4.Status/Sync_error <-> AI Standard Channel 4/Status/Sync error
//     PlcTask Inputs/GVL_iXlinker.Device_4_EtherCAT.Term_14_EK1100.Term_16_EK1122.Term_17_EK1100.Term_18_EL3174_0002.AI_Standard_Channel_1.Status/TxPDO_State <-> AI Standard Channel 1/Status/TxPDO State
//     PlcTask Inputs/GVL_iXlinker.Device_4_EtherCAT.Term_14_EK1100.Term_16_EK1122.Term_17_EK1100.Term_18_EL3174_0002.AI_Standard_Channel_2.Status/TxPDO_State <-> AI Standard Channel 2/Status/TxPDO State
//     PlcTask Inputs/GVL_iXlinker.Device_4_EtherCAT.Term_14_EK1100.Term_16_EK1122.Term_17_EK1100.Term_18_EL3174_0002.AI_Standard_Channel_3.Status/TxPDO_State <-> AI Standard Channel 3/Status/TxPDO State
//     PlcTask Inputs/GVL_iXlinker.Device_4_EtherCAT.Term_14_EK1100.Term_16_EK1122.Term_17_EK1100.Term_18_EL3174_0002.AI_Standard_Channel_4.Status/TxPDO_State <-> AI Standard Channel 4/Status/TxPDO State
//     PlcTask Inputs/GVL_iXlinker.Device_4_EtherCAT.Term_14_EK1100.Term_16_EK1122.Term_17_EK1100.Term_18_EL3174_0002.AI_Standard_Channel_1.Status/TxPDO_Toggle <-> AI Standard Channel 1/Status/TxPDO Toggle
//     PlcTask Inputs/GVL_iXlinker.Device_4_EtherCAT.Term_14_EK1100.Term_16_EK1122.Term_17_EK1100.Term_18_EL3174_0002.AI_Standard_Channel_2.Status/TxPDO_Toggle <-> AI Standard Channel 2/Status/TxPDO Toggle
//     PlcTask Inputs/GVL_iXlinker.Device_4_EtherCAT.Term_14_EK1100.Term_16_EK1122.Term_17_EK1100.Term_18_EL3174_0002.AI_Standard_Channel_3.Status/TxPDO_Toggle <-> AI Standard Channel 3/Status/TxPDO Toggle
//     PlcTask Inputs/GVL_iXlinker.Device_4_EtherCAT.Term_14_EK1100.Term_16_EK1122.Term_17_EK1100.Term_18_EL3174_0002.AI_Standard_Channel_4.Status/TxPDO_Toggle <-> AI Standard Channel 4/Status/TxPDO Toggle
//     PlcTask Inputs/GVL_iXlinker.Device_4_EtherCAT.Term_14_EK1100.Term_16_EK1122.Term_17_EK1100.Term_18_EL3174_0002.AI_Standard_Channel_1.Status/Underrange <-> AI Standard Channel 1/Status/Underrange
//     PlcTask Inputs/GVL_iXlinker.Device_4_EtherCAT.Term_14_EK1100.Term_16_EK1122.Term_17_EK1100.Term_18_EL3174_0002.AI_Standard_Channel_2.Status/Underrange <-> AI Standard Channel 2/Status/Underrange
//     PlcTask Inputs/GVL_iXlinker.Device_4_EtherCAT.Term_14_EK1100.Term_16_EK1122.Term_17_EK1100.Term_18_EL3174_0002.AI_Standard_Channel_3.Status/Underrange <-> AI Standard Channel 3/Status/Underrange
//     PlcTask Inputs/GVL_iXlinker.Device_4_EtherCAT.Term_14_EK1100.Term_16_EK1122.Term_17_EK1100.Term_18_EL3174_0002.AI_Standard_Channel_4.Status/Underrange <-> AI Standard Channel 4/Status/Underrange
//     PlcTask Inputs/GVL_iXlinker.Device_4_EtherCAT.Term_14_EK1100.Term_16_EK1122.Term_17_EK1100.Term_18_EL3174_0002.AI_Standard_Channel_1.Value <-> AI Standard Channel 1/Value
//     PlcTask Inputs/GVL_iXlinker.Device_4_EtherCAT.Term_14_EK1100.Term_16_EK1122.Term_17_EK1100.Term_18_EL3174_0002.AI_Standard_Channel_2.Value <-> AI Standard Channel 2/Value
//     PlcTask Inputs/GVL_iXlinker.Device_4_EtherCAT.Term_14_EK1100.Term_16_EK1122.Term_17_EK1100.Term_18_EL3174_0002.AI_Standard_Channel_3.Value <-> AI Standard Channel 3/Value
//     PlcTask Inputs/GVL_iXlinker.Device_4_EtherCAT.Term_14_EK1100.Term_16_EK1122.Term_17_EK1100.Term_18_EL3174_0002.AI_Standard_Channel_4.Value <-> AI Standard Channel 4/Value
//     PlcTask Inputs/GVL_iXlinker.Device_4_EtherCAT.Term_14_EK1100.Term_16_EK1122.Term_17_EK1100.Term_18_EL3174_0002.InfoData.AdsAddr <-> InfoData/AdsAddr
//     PlcTask Inputs/GVL_iXlinker.Device_4_EtherCAT.Term_14_EK1100.Term_16_EK1122.Term_17_EK1100.Term_18_EL3174_0002.InfoData.ObjectId <-> InfoData/ObjectId
//     PlcTask Inputs/GVL_iXlinker.Device_4_EtherCAT.Term_14_EK1100.Term_16_EK1122.Term_17_EK1100.Term_18_EL3174_0002.InfoData.State <-> InfoData/State
//     PlcTask Inputs/GVL_iXlinker.Device_4_EtherCAT.Term_14_EK1100.Term_16_EK1122.Term_17_EK1100.Term_18_EL3174_0002.WcState.InputToggle <-> WcState/InputToggle
//     PlcTask Inputs/GVL_iXlinker.Device_4_EtherCAT.Term_14_EK1100.Term_16_EK1122.Term_17_EK1100.Term_18_EL3174_0002.WcState.WcState <-> WcState/WcState
//   TcoIoBeckhoffTests/TcoIoBeckhoffTests Instance <-> Device 4 (EtherCAT)/Term 14 (EK1100)/Term 16 (EK1122)/Term 17 (EK1100)/Term 19 (EL6001)
//     PlcTask Inputs/GVL_iXlinker.Device_4_EtherCAT.Term_14_EK1100.Term_16_EK1122.Term_17_EK1100.Term_19_EL6001.COM_Inputs.Data_In[{0..21}] <-> COM Inputs/Data In {0..21}  (22 links)
//     PlcTask Inputs/GVL_iXlinker.Device_4_EtherCAT.Term_14_EK1100.Term_16_EK1122.Term_17_EK1100.Term_19_EL6001.COM_Inputs.Status/Buffer_full <-> COM Inputs/Status/Buffer full
//     PlcTask Inputs/GVL_iXlinker.Device_4_EtherCAT.Term_14_EK1100.Term_16_EK1122.Term_17_EK1100.Term_19_EL6001.COM_Inputs.Status/Framing_error <-> COM Inputs/Status/Framing error
//     PlcTask Inputs/GVL_iXlinker.Device_4_EtherCAT.Term_14_EK1100.Term_16_EK1122.Term_17_EK1100.Term_19_EL6001.COM_Inputs.Status/Init_accepted <-> COM Inputs/Status/Init accepted
//     PlcTask Inputs/GVL_iXlinker.Device_4_EtherCAT.Term_14_EK1100.Term_16_EK1122.Term_17_EK1100.Term_19_EL6001.COM_Inputs.Status/Input_length <-> COM Inputs/Status/Input length
//     PlcTask Inputs/GVL_iXlinker.Device_4_EtherCAT.Term_14_EK1100.Term_16_EK1122.Term_17_EK1100.Term_19_EL6001.COM_Inputs.Status/Overrun_error <-> COM Inputs/Status/Overrun error
//     PlcTask Inputs/GVL_iXlinker.Device_4_EtherCAT.Term_14_EK1100.Term_16_EK1122.Term_17_EK1100.Term_19_EL6001.COM_Inputs.Status/Parity_error <-> COM Inputs/Status/Parity error
//     PlcTask Inputs/GVL_iXlinker.Device_4_EtherCAT.Term_14_EK1100.Term_16_EK1122.Term_17_EK1100.Term_19_EL6001.COM_Inputs.Status/Receive_request <-> COM Inputs/Status/Receive request
//     PlcTask Inputs/GVL_iXlinker.Device_4_EtherCAT.Term_14_EK1100.Term_16_EK1122.Term_17_EK1100.Term_19_EL6001.COM_Inputs.Status/Transmit_accepted <-> COM Inputs/Status/Transmit accepted
//     PlcTask Inputs/GVL_iXlinker.Device_4_EtherCAT.Term_14_EK1100.Term_16_EK1122.Term_17_EK1100.Term_19_EL6001.InfoData.AdsAddr <-> InfoData/AdsAddr
//     PlcTask Inputs/GVL_iXlinker.Device_4_EtherCAT.Term_14_EK1100.Term_16_EK1122.Term_17_EK1100.Term_19_EL6001.InfoData.ObjectId <-> InfoData/ObjectId
//     PlcTask Inputs/GVL_iXlinker.Device_4_EtherCAT.Term_14_EK1100.Term_16_EK1122.Term_17_EK1100.Term_19_EL6001.InfoData.State <-> InfoData/State
//     PlcTask Inputs/GVL_iXlinker.Device_4_EtherCAT.Term_14_EK1100.Term_16_EK1122.Term_17_EK1100.Term_19_EL6001.WcState.InputToggle <-> WcState/InputToggle
//     PlcTask Inputs/GVL_iXlinker.Device_4_EtherCAT.Term_14_EK1100.Term_16_EK1122.Term_17_EK1100.Term_19_EL6001.WcState.WcState <-> WcState/WcState
//     PlcTask Outputs/GVL_iXlinker.Device_4_EtherCAT.Term_14_EK1100.Term_16_EK1122.Term_17_EK1100.Term_19_EL6001.COM_Outputs.Ctrl/Init_request <-> COM Outputs/Ctrl/Init request
//     PlcTask Outputs/GVL_iXlinker.Device_4_EtherCAT.Term_14_EK1100.Term_16_EK1122.Term_17_EK1100.Term_19_EL6001.COM_Outputs.Ctrl/Output_length <-> COM Outputs/Ctrl/Output length
//     PlcTask Outputs/GVL_iXlinker.Device_4_EtherCAT.Term_14_EK1100.Term_16_EK1122.Term_17_EK1100.Term_19_EL6001.COM_Outputs.Ctrl/Receive_accepted <-> COM Outputs/Ctrl/Receive accepted
//     PlcTask Outputs/GVL_iXlinker.Device_4_EtherCAT.Term_14_EK1100.Term_16_EK1122.Term_17_EK1100.Term_19_EL6001.COM_Outputs.Ctrl/Send_continues <-> COM Outputs/Ctrl/Send continues
//     PlcTask Outputs/GVL_iXlinker.Device_4_EtherCAT.Term_14_EK1100.Term_16_EK1122.Term_17_EK1100.Term_19_EL6001.COM_Outputs.Ctrl/Transmit_request <-> COM Outputs/Ctrl/Transmit request
//     PlcTask Outputs/GVL_iXlinker.Device_4_EtherCAT.Term_14_EK1100.Term_16_EK1122.Term_17_EK1100.Term_19_EL6001.COM_Outputs.Data_Out[{0..21}] <-> COM Outputs/Data Out {0..21}  (22 links)
//   TcoIoBeckhoffTests/TcoIoBeckhoffTests Instance <-> Device 4 (EtherCAT)/Term 14 (EK1100)/Term 16 (EK1122)/Term 17 (EK1100)/Term 20 (EL3011)
//     PlcTask Inputs/GVL_iXlinker.Device_4_EtherCAT.Term_14_EK1100.Term_16_EK1122.Term_17_EK1100.Term_20_EL3011.AI_Standard.Status/Error <-> AI Standard/Status/Error
//     PlcTask Inputs/GVL_iXlinker.Device_4_EtherCAT.Term_14_EK1100.Term_16_EK1122.Term_17_EK1100.Term_20_EL3011.AI_Standard.Status/Limit_1 <-> AI Standard/Status/Limit 1
//     PlcTask Inputs/GVL_iXlinker.Device_4_EtherCAT.Term_14_EK1100.Term_16_EK1122.Term_17_EK1100.Term_20_EL3011.AI_Standard.Status/Limit_2 <-> AI Standard/Status/Limit 2
//     PlcTask Inputs/GVL_iXlinker.Device_4_EtherCAT.Term_14_EK1100.Term_16_EK1122.Term_17_EK1100.Term_20_EL3011.AI_Standard.Status/Overrange <-> AI Standard/Status/Overrange
//     PlcTask Inputs/GVL_iXlinker.Device_4_EtherCAT.Term_14_EK1100.Term_16_EK1122.Term_17_EK1100.Term_20_EL3011.AI_Standard.Status/TxPDO_State <-> AI Standard/Status/TxPDO State
//     PlcTask Inputs/GVL_iXlinker.Device_4_EtherCAT.Term_14_EK1100.Term_16_EK1122.Term_17_EK1100.Term_20_EL3011.AI_Standard.Status/TxPDO_Toggle <-> AI Standard/Status/TxPDO Toggle
//     PlcTask Inputs/GVL_iXlinker.Device_4_EtherCAT.Term_14_EK1100.Term_16_EK1122.Term_17_EK1100.Term_20_EL3011.AI_Standard.Status/Underrange <-> AI Standard/Status/Underrange
//     PlcTask Inputs/GVL_iXlinker.Device_4_EtherCAT.Term_14_EK1100.Term_16_EK1122.Term_17_EK1100.Term_20_EL3011.AI_Standard.Value <-> AI Standard/Value
//     PlcTask Inputs/GVL_iXlinker.Device_4_EtherCAT.Term_14_EK1100.Term_16_EK1122.Term_17_EK1100.Term_20_EL3011.InfoData.AdsAddr <-> InfoData/AdsAddr
//     PlcTask Inputs/GVL_iXlinker.Device_4_EtherCAT.Term_14_EK1100.Term_16_EK1122.Term_17_EK1100.Term_20_EL3011.InfoData.ObjectId <-> InfoData/ObjectId
//     PlcTask Inputs/GVL_iXlinker.Device_4_EtherCAT.Term_14_EK1100.Term_16_EK1122.Term_17_EK1100.Term_20_EL3011.InfoData.State <-> InfoData/State
//     PlcTask Inputs/GVL_iXlinker.Device_4_EtherCAT.Term_14_EK1100.Term_16_EK1122.Term_17_EK1100.Term_20_EL3011.WcState.InputToggle <-> WcState/InputToggle
//     PlcTask Inputs/GVL_iXlinker.Device_4_EtherCAT.Term_14_EK1100.Term_16_EK1122.Term_17_EK1100.Term_20_EL3011.WcState.WcState <-> WcState/WcState
//   TcoIoBeckhoffTests/TcoIoBeckhoffTests Instance <-> Device 4 (EtherCAT)/Term 14 (EK1100)/Term 16 (EK1122)/Term 17 (EK1100)/Term 21 (EL2008)
//     PlcTask Inputs/GVL_iXlinker.Device_4_EtherCAT.Term_14_EK1100.Term_16_EK1122.Term_17_EK1100.Term_21_EL2008.InfoData.AdsAddr <-> InfoData/AdsAddr
//     PlcTask Inputs/GVL_iXlinker.Device_4_EtherCAT.Term_14_EK1100.Term_16_EK1122.Term_17_EK1100.Term_21_EL2008.InfoData.ObjectId <-> InfoData/ObjectId
//     PlcTask Inputs/GVL_iXlinker.Device_4_EtherCAT.Term_14_EK1100.Term_16_EK1122.Term_17_EK1100.Term_21_EL2008.InfoData.State <-> InfoData/State
//     PlcTask Inputs/GVL_iXlinker.Device_4_EtherCAT.Term_14_EK1100.Term_16_EK1122.Term_17_EK1100.Term_21_EL2008.WcState.WcState <-> WcState/WcState
//     PlcTask Outputs/GVL_iXlinker.Device_4_EtherCAT.Term_14_EK1100.Term_16_EK1122.Term_17_EK1100.Term_21_EL2008.Channel_{1..8}.Output <-> Channel {1..8}/Output  (8 links)
//   TcoIoBeckhoffTests/TcoIoBeckhoffTests Instance <-> Device 4 (EtherCAT)/Term 14 (EK1100)/Term 16 (EK1122)/Term 17 (EK1100)/Term 22 (EL2008)
//     PlcTask Inputs/GVL_iXlinker.Device_4_EtherCAT.Term_14_EK1100.Term_16_EK1122.Term_17_EK1100.Term_22_EL2008.InfoData.AdsAddr <-> InfoData/AdsAddr
//     PlcTask Inputs/GVL_iXlinker.Device_4_EtherCAT.Term_14_EK1100.Term_16_EK1122.Term_17_EK1100.Term_22_EL2008.InfoData.ObjectId <-> InfoData/ObjectId
//     PlcTask Inputs/GVL_iXlinker.Device_4_EtherCAT.Term_14_EK1100.Term_16_EK1122.Term_17_EK1100.Term_22_EL2008.InfoData.State <-> InfoData/State
//     PlcTask Inputs/GVL_iXlinker.Device_4_EtherCAT.Term_14_EK1100.Term_16_EK1122.Term_17_EK1100.Term_22_EL2008.WcState.WcState <-> WcState/WcState
//     PlcTask Outputs/GVL_iXlinker.Device_4_EtherCAT.Term_14_EK1100.Term_16_EK1122.Term_17_EK1100.Term_22_EL2008.Channel_{1..8}.Output <-> Channel {1..8}/Output  (8 links)
//   TcoIoBeckhoffTests/TcoIoBeckhoffTests Instance <-> Device 4 (EtherCAT)/Term 14 (EK1100)/Term 23 (EL3024)
//     PlcTask Inputs/GVL_iXlinker.Device_4_EtherCAT.Term_14_EK1100.Term_23_EL3024.AI_Standard_Channel_{1..4}.Status/Error <-> AI Standard Channel {1..4}/Status/Error  (4 links)
//     PlcTask Inputs/GVL_iXlinker.Device_4_EtherCAT.Term_14_EK1100.Term_23_EL3024.AI_Standard_Channel_1.Status/Limit_1 <-> AI Standard Channel 1/Status/Limit 1
//     PlcTask Inputs/GVL_iXlinker.Device_4_EtherCAT.Term_14_EK1100.Term_23_EL3024.AI_Standard_Channel_1.Status/Limit_2 <-> AI Standard Channel 1/Status/Limit 2
//     PlcTask Inputs/GVL_iXlinker.Device_4_EtherCAT.Term_14_EK1100.Term_23_EL3024.AI_Standard_Channel_2.Status/Limit_1 <-> AI Standard Channel 2/Status/Limit 1
//     PlcTask Inputs/GVL_iXlinker.Device_4_EtherCAT.Term_14_EK1100.Term_23_EL3024.AI_Standard_Channel_2.Status/Limit_2 <-> AI Standard Channel 2/Status/Limit 2
//     PlcTask Inputs/GVL_iXlinker.Device_4_EtherCAT.Term_14_EK1100.Term_23_EL3024.AI_Standard_Channel_3.Status/Limit_1 <-> AI Standard Channel 3/Status/Limit 1
//     PlcTask Inputs/GVL_iXlinker.Device_4_EtherCAT.Term_14_EK1100.Term_23_EL3024.AI_Standard_Channel_3.Status/Limit_2 <-> AI Standard Channel 3/Status/Limit 2
//     PlcTask Inputs/GVL_iXlinker.Device_4_EtherCAT.Term_14_EK1100.Term_23_EL3024.AI_Standard_Channel_4.Status/Limit_1 <-> AI Standard Channel 4/Status/Limit 1
//     PlcTask Inputs/GVL_iXlinker.Device_4_EtherCAT.Term_14_EK1100.Term_23_EL3024.AI_Standard_Channel_4.Status/Limit_2 <-> AI Standard Channel 4/Status/Limit 2
//     PlcTask Inputs/GVL_iXlinker.Device_4_EtherCAT.Term_14_EK1100.Term_23_EL3024.AI_Standard_Channel_{1..4}.Status/Overrange <-> AI Standard Channel {1..4}/Status/Overrange  (4 links)
//     PlcTask Inputs/GVL_iXlinker.Device_4_EtherCAT.Term_14_EK1100.Term_23_EL3024.AI_Standard_Channel_{1..4}.Status/TxPDO_State <-> AI Standard Channel {1..4}/Status/TxPDO State  (4 links)
//     PlcTask Inputs/GVL_iXlinker.Device_4_EtherCAT.Term_14_EK1100.Term_23_EL3024.AI_Standard_Channel_{1..4}.Status/TxPDO_Toggle <-> AI Standard Channel {1..4}/Status/TxPDO Toggle  (4 links)
//     PlcTask Inputs/GVL_iXlinker.Device_4_EtherCAT.Term_14_EK1100.Term_23_EL3024.AI_Standard_Channel_{1..4}.Status/Underrange <-> AI Standard Channel {1..4}/Status/Underrange  (4 links)
//     PlcTask Inputs/GVL_iXlinker.Device_4_EtherCAT.Term_14_EK1100.Term_23_EL3024.AI_Standard_Channel_{1..4}.Value <-> AI Standard Channel {1..4}/Value  (4 links)
//     PlcTask Inputs/GVL_iXlinker.Device_4_EtherCAT.Term_14_EK1100.Term_23_EL3024.InfoData.AdsAddr <-> InfoData/AdsAddr
//     PlcTask Inputs/GVL_iXlinker.Device_4_EtherCAT.Term_14_EK1100.Term_23_EL3024.InfoData.ObjectId <-> InfoData/ObjectId
//     PlcTask Inputs/GVL_iXlinker.Device_4_EtherCAT.Term_14_EK1100.Term_23_EL3024.InfoData.State <-> InfoData/State
//     PlcTask Inputs/GVL_iXlinker.Device_4_EtherCAT.Term_14_EK1100.Term_23_EL3024.WcState.InputToggle <-> WcState/InputToggle
//     PlcTask Inputs/GVL_iXlinker.Device_4_EtherCAT.Term_14_EK1100.Term_23_EL3024.WcState.WcState <-> WcState/WcState
//   TcoIoBeckhoffTests/TcoIoBeckhoffTests Instance <-> Device 4 (EtherCAT)/Term 9 (EK1100)
//     PlcTask Inputs/GVL_iXlinker.Device_4_EtherCAT.Term_9_EK1100.InfoData.AdsAddr <-> InfoData/AdsAddr
//     PlcTask Inputs/GVL_iXlinker.Device_4_EtherCAT.Term_9_EK1100.InfoData.ObjectId <-> InfoData/ObjectId
//     PlcTask Inputs/GVL_iXlinker.Device_4_EtherCAT.Term_9_EK1100.InfoData.State <-> InfoData/State
//   TcoIoBeckhoffTests/TcoIoBeckhoffTests Instance <-> Device 4 (EtherCAT)/Term 9 (EK1100)/Term 10 (EL6001)
//     PlcTask Inputs/GVL_iXlinker.Device_4_EtherCAT.Term_9_EK1100.Term_10_EL6001.COM_Inputs.Data_In[{0..21}] <-> COM Inputs/Data In {0..21}  (22 links)
//     PlcTask Inputs/GVL_iXlinker.Device_4_EtherCAT.Term_9_EK1100.Term_10_EL6001.COM_Inputs.Status/Buffer_full <-> COM Inputs/Status/Buffer full
//     PlcTask Inputs/GVL_iXlinker.Device_4_EtherCAT.Term_9_EK1100.Term_10_EL6001.COM_Inputs.Status/Framing_error <-> COM Inputs/Status/Framing error
//     PlcTask Inputs/GVL_iXlinker.Device_4_EtherCAT.Term_9_EK1100.Term_10_EL6001.COM_Inputs.Status/Init_accepted <-> COM Inputs/Status/Init accepted
//     PlcTask Inputs/GVL_iXlinker.Device_4_EtherCAT.Term_9_EK1100.Term_10_EL6001.COM_Inputs.Status/Input_length <-> COM Inputs/Status/Input length
//     PlcTask Inputs/GVL_iXlinker.Device_4_EtherCAT.Term_9_EK1100.Term_10_EL6001.COM_Inputs.Status/Overrun_error <-> COM Inputs/Status/Overrun error
//     PlcTask Inputs/GVL_iXlinker.Device_4_EtherCAT.Term_9_EK1100.Term_10_EL6001.COM_Inputs.Status/Parity_error <-> COM Inputs/Status/Parity error
//     PlcTask Inputs/GVL_iXlinker.Device_4_EtherCAT.Term_9_EK1100.Term_10_EL6001.COM_Inputs.Status/Receive_request <-> COM Inputs/Status/Receive request
//     PlcTask Inputs/GVL_iXlinker.Device_4_EtherCAT.Term_9_EK1100.Term_10_EL6001.COM_Inputs.Status/Transmit_accepted <-> COM Inputs/Status/Transmit accepted
//     PlcTask Inputs/GVL_iXlinker.Device_4_EtherCAT.Term_9_EK1100.Term_10_EL6001.InfoData.AdsAddr <-> InfoData/AdsAddr
//     PlcTask Inputs/GVL_iXlinker.Device_4_EtherCAT.Term_9_EK1100.Term_10_EL6001.InfoData.ObjectId <-> InfoData/ObjectId
//     PlcTask Inputs/GVL_iXlinker.Device_4_EtherCAT.Term_9_EK1100.Term_10_EL6001.InfoData.State <-> InfoData/State
//     PlcTask Inputs/GVL_iXlinker.Device_4_EtherCAT.Term_9_EK1100.Term_10_EL6001.WcState.InputToggle <-> WcState/InputToggle
//     PlcTask Inputs/GVL_iXlinker.Device_4_EtherCAT.Term_9_EK1100.Term_10_EL6001.WcState.WcState <-> WcState/WcState
//     PlcTask Outputs/GVL_iXlinker.Device_4_EtherCAT.Term_9_EK1100.Term_10_EL6001.COM_Outputs.Ctrl/Init_request <-> COM Outputs/Ctrl/Init request
//     PlcTask Outputs/GVL_iXlinker.Device_4_EtherCAT.Term_9_EK1100.Term_10_EL6001.COM_Outputs.Ctrl/Output_length <-> COM Outputs/Ctrl/Output length
//     PlcTask Outputs/GVL_iXlinker.Device_4_EtherCAT.Term_9_EK1100.Term_10_EL6001.COM_Outputs.Ctrl/Receive_accepted <-> COM Outputs/Ctrl/Receive accepted
//     PlcTask Outputs/GVL_iXlinker.Device_4_EtherCAT.Term_9_EK1100.Term_10_EL6001.COM_Outputs.Ctrl/Send_continues <-> COM Outputs/Ctrl/Send continues
//     PlcTask Outputs/GVL_iXlinker.Device_4_EtherCAT.Term_9_EK1100.Term_10_EL6001.COM_Outputs.Ctrl/Transmit_request <-> COM Outputs/Ctrl/Transmit request
//     PlcTask Outputs/GVL_iXlinker.Device_4_EtherCAT.Term_9_EK1100.Term_10_EL6001.COM_Outputs.Data_Out[{0..21}] <-> COM Outputs/Data Out {0..21}  (22 links)
//   TcoIoBeckhoffTests/TcoIoBeckhoffTests Instance <-> Device 4 (EtherCAT)/Term 9 (EK1100)/Term 11 (EL1809)
//     PlcTask Inputs/GVL_iXlinker.Device_4_EtherCAT.Term_9_EK1100.Term_11_EL1809.Channel_{1..16}.Input <-> Channel {1..16}/Input  (16 links)
//     PlcTask Inputs/GVL_iXlinker.Device_4_EtherCAT.Term_9_EK1100.Term_11_EL1809.InfoData.AdsAddr <-> InfoData/AdsAddr
//     PlcTask Inputs/GVL_iXlinker.Device_4_EtherCAT.Term_9_EK1100.Term_11_EL1809.InfoData.ObjectId <-> InfoData/ObjectId
//     PlcTask Inputs/GVL_iXlinker.Device_4_EtherCAT.Term_9_EK1100.Term_11_EL1809.InfoData.State <-> InfoData/State
//     PlcTask Inputs/GVL_iXlinker.Device_4_EtherCAT.Term_9_EK1100.Term_11_EL1809.WcState.InputToggle <-> WcState/InputToggle
//     PlcTask Inputs/GVL_iXlinker.Device_4_EtherCAT.Term_9_EK1100.Term_11_EL1809.WcState.WcState <-> WcState/WcState
//   TcoIoBeckhoffTests/TcoIoBeckhoffTests Instance <-> Device 4 (EtherCAT)/Term 9 (EK1100)/Term 12 (EL2809)
//     PlcTask Inputs/GVL_iXlinker.Device_4_EtherCAT.Term_9_EK1100.Term_12_EL2809.InfoData.AdsAddr <-> InfoData/AdsAddr
//     PlcTask Inputs/GVL_iXlinker.Device_4_EtherCAT.Term_9_EK1100.Term_12_EL2809.InfoData.ObjectId <-> InfoData/ObjectId
//     PlcTask Inputs/GVL_iXlinker.Device_4_EtherCAT.Term_9_EK1100.Term_12_EL2809.InfoData.State <-> InfoData/State
//     PlcTask Inputs/GVL_iXlinker.Device_4_EtherCAT.Term_9_EK1100.Term_12_EL2809.WcState.WcState <-> WcState/WcState
//     PlcTask Outputs/GVL_iXlinker.Device_4_EtherCAT.Term_9_EK1100.Term_12_EL2809.Channel_{1..16}.Output <-> Channel {1..16}/Output  (16 links)
//   TcoIoBeckhoffTests/TcoIoBeckhoffTests Instance <-> Device 4 (EtherCAT)/Term 9 (EK1100)/Term 13 (EK1110)
//     PlcTask Inputs/GVL_iXlinker.Device_4_EtherCAT.Term_9_EK1100.Term_13_EK1110.InfoData.AdsAddr <-> InfoData/AdsAddr
//     PlcTask Inputs/GVL_iXlinker.Device_4_EtherCAT.Term_9_EK1100.Term_13_EK1110.InfoData.ObjectId <-> InfoData/ObjectId
//     PlcTask Inputs/GVL_iXlinker.Device_4_EtherCAT.Term_9_EK1100.Term_13_EK1110.InfoData.State <-> InfoData/State

// ---- Diagnostics/EtherCAT/MasterDevice/TcoEthercatDiagnosticsTask.TcPOU
FUNCTION_BLOCK TcoEthercatDiagnosticsTask EXTENDS TcoCore.TcoTask
VAR_INPUT
	inNetId : Tc2_System.T_AmsNetID;
END_VAR
VAR
    _EcGetAllSlaveStates 	: Tc2_EtherCAT.FB_EcGetAllSlaveStates;
    _EcGetConfSlaves 		: Tc2_EtherCAT.FB_EcGetConfSlaves;
	_updateDiagnosticsState : TcoCore.TcoState(THIS^,TcoCore.eRestoreMode.None);

	_SlaveStatesCount      		: UINT;
    _ConfigSlavesCount     		: UINT;
    _SlaveStateBuffer      		: ARRAY[0..EC_MAX_SLAVES] OF Tc2_EtherCAT.ST_EcSlaveState;
    _SlaveConfigDataBuffer 		: ARRAY[0..EC_MAX_SLAVES] OF Tc2_EtherCAT.ST_EcSlaveConfigData;

	_i	:	UINT;

	_name : STRING;
	_type : STRING;
	_state : STRING;
	
	_DiagnosticsMessengers		: DiagnosticsMessengers(THIS^);
	_DiagnosticsMessengerIndex	: UINT;	
END_VAR
VAR_OUTPUT
	outDiagnosticsAvailable : BOOL;
END_VAR

IF Execute() THEN
	IF _updateDiagnosticsState.State = 10 THEN
		outDiagnosticsAvailable := FALSE;
		_EcGetAllSlaveStates(bExecute := FALSE);
		_EcGetConfSlaves(bExecute := FALSE);
	
		IF NOT _EcGetAllSlaveStates.bBusy AND NOT _EcGetAllSlaveStates.bError AND NOT _EcGetConfSlaves.bBusy AND NOT _EcGetConfSlaves.bError THEN
			_updateDiagnosticsState.ChangeState(_updateDiagnosticsState._State + 10);
		END_IF
	END_IF
	
	IF _updateDiagnosticsState.State = 20 THEN
		_EcGetAllSlaveStates(sNetId := inNetId,
			pStateBuf := ADR(_SlaveStateBuffer),
			cbBufLen := SIZEOF(_SlaveStateBuffer),
			bExecute := TRUE,
			tTimeout :=,
			bBusy =>,
			bError =>,
			nErrId =>,
			nSlaves => _SlaveStatesCount);
	
		IF _EcGetAllSlaveStates.bBusy THEN
			_updateDiagnosticsState.ChangeState(_updateDiagnosticsState._State + 10);
		END_IF
	END_IF
	
	IF _updateDiagnosticsState.State = 30 THEN
		_EcGetAllSlaveStates(sNetId := inNetId,
			pStateBuf := ADR(_SlaveStateBuffer),
			cbBufLen := SIZEOF(_SlaveStateBuffer),
			bExecute := FALSE,
			tTimeout :=,
			bBusy =>,
			bError =>,
			nErrId =>,
			nSlaves => _SlaveStatesCount);
	
		IF NOT _EcGetAllSlaveStates.bBusy AND NOT _EcGetAllSlaveStates.bError THEN
			_updateDiagnosticsState.ChangeState(_updateDiagnosticsState._State + 10);
		END_IF
	END_IF
	
	IF _updateDiagnosticsState.State = 40 THEN
		_EcGetConfSlaves(sNetId := inNetId,
			pArrEcConfSlaveInfo := ADR(_SlaveConfigDataBuffer),
			cbBufLen := SIZEOF(_SlaveConfigDataBuffer),
			bExecute := TRUE,
			tTimeout :=,
			bBusy =>,
			bError =>,
			nErrorId =>,
			nSlaves => _ConfigSlavesCount);
	
		IF _EcGetConfSlaves.bBusy THEN
			_updateDiagnosticsState.ChangeState(_updateDiagnosticsState._State + 10);
		END_IF
	END_IF
	
	IF _updateDiagnosticsState.State = 50 THEN
		_EcGetConfSlaves(sNetId := inNetId,
			pArrEcConfSlaveInfo := ADR(_SlaveConfigDataBuffer),
			cbBufLen := SIZEOF(_SlaveConfigDataBuffer),
			bExecute := FALSE,
			tTimeout :=,
			bBusy =>,
			bError =>,
			nErrorId =>,
			nSlaves => _ConfigSlavesCount);
	
		IF NOT _EcGetConfSlaves.bBusy AND NOT _EcGetConfSlaves.bError THEN
			_updateDiagnosticsState.ChangeState(_updateDiagnosticsState._State + 10);
		END_IF
	END_IF
	
	IF _updateDiagnosticsState.State = 60 THEN
		_EcGetAllSlaveStates(bExecute := FALSE);
		_EcGetConfSlaves(bExecute := FALSE);
	
		IF NOT _EcGetAllSlaveStates.bBusy AND NOT _EcGetAllSlaveStates.bError AND NOT _EcGetConfSlaves.bBusy AND NOT _EcGetConfSlaves.bError THEN
			_updateDiagnosticsState.ChangeState(_updateDiagnosticsState._State + 10);
		END_IF
	END_IF
	
	IF _updateDiagnosticsState.State = 70 THEN
		_DiagnosticsMessengerIndex := 0;
	    FOR _i := 0 TO _ConfigSlavesCount DO
			IF (_SlaveStateBuffer[_i].deviceState <> 8 OR _SlaveStateBuffer[_i].linkState <> 0) THEN
				IF _SlaveConfigDataBuffer[_i].sName <> '' THEN
					IF _DiagnosticsMessengerIndex <= 2 THEN
						outDiagnosticsAvailable := TRUE;
						_name := _SlaveConfigDataBuffer[_i].sName;
						_type := Tc2_EtherCAT.F_ConvProductCodeToString(_SlaveConfigDataBuffer[_i].stSlaveIdentity);
						_state :=  Tc2_EtherCAT.F_ConvSlaveStateToString(state := _SlaveStateBuffer[_i]);
						_DiagnosticsMessengers.Messengers[_DiagnosticsMessengerIndex].Build().AppendAny(_name).Append('[').AppendAny(_type).Append(']').Append( _state).As().AsError().Pin();
						_DiagnosticsMessengerIndex := _DiagnosticsMessengerIndex + 1;
					END_IF
				END_IF
			END_IF;
	    END_FOR

		_updateDiagnosticsState.ChangeState(_updateDiagnosticsState._State + 10);
	END_IF
	
	IF _updateDiagnosticsState.State = 80 THEN
		DoneWhen(TRUE);
	END_IF

	ThrowWhen(_EcGetAllSlaveStates.bError OR _EcGetConfSlaves.bError);
END_IF

(*~
	<docu>
		<summary>
			Executes when task is aborted.
		</summary>			
	</docu>	
~*)
METHOD PROTECTED OnAbort
_EcGetAllSlaveStates(bExecute := FALSE);
_EcGetConfSlaves(bExecute := FALSE);

_updateDiagnosticsState.Restore();
END_METHOD

(*~
	<docu>
		<summary>
			Executes when task reaches the ```Done``` state .
		</summary>			
	</docu>	
~*)
METHOD PROTECTED OnDone
_EcGetAllSlaveStates(bExecute := FALSE);
_EcGetConfSlaves(bExecute := FALSE);
END_METHOD

(*~
	<docu>
		<summary>
			Executes when task reaches the ```Error``` state.
			<para>
				Do not confuse with <see cref="PlcDocu.TcoCore.TcoTask.WhileError()"/>, that is called cyclically until '''Error''' state is left.
			</para>
		</summary>			
	</docu>	
~*)
METHOD PROTECTED OnError
IF _EcGetAllSlaveStates.bError THEN
	Messenger.Build().Append('Reading status of all EtherCAT slaves using "Tc2_EtherCAT.FB_EcGetAllSlaveStates" function block returns error. nErrId: ').AppendAny(_EcGetAllSlaveStates.nErrId).As().AsError();
ELSIF _EcGetConfSlaves.bError THEN
	Messenger.Build().Append('Reading status of configurateed EtherCAT slaves using "Tc2_EtherCAT.FB_EcGetConfSlaves" function block returns error. nErrorId: ').AppendAny(_EcGetConfSlaves.nErrorId).As().AsError();
END_IF
END_METHOD

METHOD PROTECTED OnStart
_EcGetAllSlaveStates(bExecute := FALSE);
_EcGetConfSlaves(bExecute := FALSE);

_updateDiagnosticsState.ChangeState(10);
END_METHOD

(*~
	<docu>
		<summary>
			Restores this instance to the Ready state. Can be called explicitly or from within one of the restore mechanisms.
			<para>
				See also <see cref="PlcDocu.TcoCore.TcoTask.AutoRestorable()"/>
			</para>
		</summary>			
	</docu>	
~*)
METHOD Restore : ITcoRestorable
THIS^._EcGetAllSlaveStates(bExecute := FALSE);
THIS^._EcGetConfSlaves(bExecute := FALSE);

THIS^._DiagnosticsMessengers.Messengers[0].Clear();
THIS^._DiagnosticsMessengers.Messengers[1].Clear();
THIS^._DiagnosticsMessengers.Messengers[2].Clear();

THIS^.outDiagnosticsAvailable := FALSE;
THIS^._updateDiagnosticsState.Restore();

SUPER^.Restore();
END_METHOD

END_FUNCTION_BLOCK

// ---- Diagnostics/EtherCAT/MasterDevice/TcoEthercatMasterDevice.TcPOU
FUNCTION_BLOCK TcoEthercatMasterDevice EXTENDS TcoCore.TcoComponent IMPLEMENTS ITcoEthercatMasterDevice
VAR_INPUT
    Inputs   		:	Inputs_5FC39E3C;
    InfoData		:	InfoData_45F98C50;
	SyncUnits		:	POINTER TO SyncUnitTask_B4157F22;
	SyncUnitsSize	:	UINT;
END_VAR

VAR
    _someSyncUnitHasSomeIssue	: BOOL;
    _allDataValid          		: BOOL;
    _someDataInvalid       		: BOOL;
    _State                		: TcoEthercatMasterDeviceState;
    _NetId                 		: Tc2_System.T_AmsNetID;
    _DeviceHasSomeIssue    		: BOOL;
    _TcoEthercatDiagnosticsTask	: TcoEthercatDiagnosticsTask(THIS^);

    _InfoDataChangeCountPV 		: UINT;

	_numberOfSyncUnits			: UINT;

	{attribute addProperty Name "Acknowledge"}
	_acknowledge				:	TcoCore.TcoTask(THIS^);
	
	_DiagnosticsAvailable : BOOL;
END_VAR
VAR_OUTPUT
    Outputs  : Outputs_C46FA7B3;
END_VAR

UpdateSyncUnitsStatus(SyncUnits,SyncUnitsSize);
Diagnostics();

PROPERTY AllDataValid : BOOL
GET
AllDataValid := _allDataValid;
END_GET
END_PROPERTY

PROPERTY DeviceHasSomeIssue : BOOL
GET
_DeviceHasSomeIssue		:=	_State.LinkError							 	OR
							_State.IOLockedAfterLinkError 					OR
							_State.LinkErrorRedundancyAdapter	 			OR
							_State.MissingOneFrame 							OR
							_State.OutOfSendResources 						OR
							_State.WatchdogTriggered 						OR
							_State.EthernetDriverNotFound 					OR
							_State.IOResetActive 							OR
							_State.AtLeastOneDeviceInInitState 				OR
							_State.AtLeastOneDeviceInPreOpState 			OR
							_State.AtLeastOneDeviceInSafeOpState 			OR
							_State.AtLeastOneDeviceIndicatesAnErrorState 	OR
							_State.DcNotInSync 								;
							
DeviceHasSomeIssue := _DeviceHasSomeIssue;
END_GET
END_PROPERTY

METHOD Diagnostics
VAR
    _i : UINT;
END_VAR
_NetId := Tc2_System.F_CreateAmsNetId(InfoData.AmsNetId);

_TcoEthercatDiagnosticsTask(inNetId := _NetId, outDiagnosticsAvailable => _DiagnosticsAvailable);

Service();

IF _acknowledge.Execute() THEN
	Restore();	
END_IF

IF (DeviceHasSomeIssue OR SomeSyncUnitHasSomeIssue OR SomeDataInvalid OR _InfoDataChangeCountPV <> InfoData.ChangeCount) (*OR _manualDiagnosticStart.Execute()*) THEN
	IF _TcoEthercatDiagnosticsTask.Ready THEN
		_InfoDataChangeCountPV := InfoData.ChangeCount;
		_TcoEthercatDiagnosticsTask.Invoke();
	END_IF
	IF _TcoEthercatDiagnosticsTask.Done AND NOT _DiagnosticsAvailable THEN
		_TcoEthercatDiagnosticsTask.Restore();
	END_IF;
END_IF
END_METHOD

METHOD FB_init : BOOL
VAR_INPUT
	bInitRetains : BOOL; // if TRUE, the retain variables are initialized (warm start / cold start)
	bInCopyCode : BOOL;  // if TRUE, the instance afterwards gets moved into the copy code (online change)
	ParentObject : TcoCore.ITcoObject;	
END_VAR
END_METHOD

(*~
	<docu>
		<summary>
			Restores this instance to the Ready state. Can be called explicitly or from within one of the restore mechanisms.	
		</summary>			
	</docu>	
~*)
METHOD  Restore : ITcoRestorable
THIS^.Messenger.Clear();
THIS^._DiagnosticsAvailable := FALSE;
THIS^._acknowledge.Restore();
THIS^._TcoEthercatDiagnosticsTask.Restore();
END_METHOD

(*~
	<docu>
		<summary>
		    Custom service (manual, maintenance) logic.
			This method must be implemented in derived class.
		</summary>			
	</docu>	
~*)
METHOD PROTECTED  ServiceMode
_acknowledge();
END_METHOD

PROPERTY SomeDataInvalid : BOOL
GET
SomeDataInvalid := _someDataInvalid;
END_GET
END_PROPERTY

PROPERTY SomeSyncUnitHasSomeIssue : BOOL
GET
SomeSyncUnitHasSomeIssue := _someSyncUnitHasSomeIssue;
END_GET
END_PROPERTY

PROPERTY State : TcoEthercatMasterDeviceState
GET
_State.LinkError							 	:= Inputs.DevState.0;
_State.IOLockedAfterLinkError 					:= Inputs.DevState.1;
_State.LinkErrorRedundancyAdapter	 			:= Inputs.DevState.2;
_State.MissingOneFrame 							:= Inputs.DevState.3;
_State.OutOfSendResources 						:= Inputs.DevState.4;
_State.WatchdogTriggered 						:= Inputs.DevState.5;
_State.EthernetDriverNotFound 					:= Inputs.DevState.6;
_State.IOResetActive 							:= Inputs.DevState.7;
_State.AtLeastOneDeviceInInitState 				:= Inputs.DevState.8;
_State.AtLeastOneDeviceInPreOpState 			:= Inputs.DevState.9;
_State.AtLeastOneDeviceInSafeOpState 			:= Inputs.DevState.10;
_State.AtLeastOneDeviceIndicatesAnErrorState 	:= Inputs.DevState.11;
_State.DcNotInSync 								:= Inputs.DevState.12;

State := _State;
END_GET
END_PROPERTY

METHOD SyncUnitHasSomeIssue : BOOL
VAR_INPUT
	inState : UINT;
END_VAR
VAR
	_state : SyncUnitState;
END_VAR
_state.AtLeastOneSlaveInInitState 				:=	inState.0 AND NOT	inState.1;
_state.AtLeastOneSlaveInPreopState 				:=	inState.0 AND 		inState.1;
_state.AtLeastOneSlaveInBootState 				:=	inState.0 AND		inState.1;
_state.AtLeastOneSlaveInSafeOpState 			:=	inState.2;
_state.AtLeastOneSlaveInOpState 				:=	inState.3;
_state.AtLeastOneSlaveSignalsError 				:=	inState.4;
_state.InvalidVendoridOrProductcodeRead 		:=	inState.5;
_state.InitializationErrorOccurred				:=	inState.6;
_state.AtLeastOneSlaveDisabled					:=	inState.7;
_state.AtLeastOneSlaveNotPresent				:=	inState.8;
_state.AtLeastOneSlaveSignalsLinkError			:=	inState.9;
_state.AtLeastOneSlaveSignalsMissingLink		:=	inState.10;
_state.AtLeastOneSlaveSignalsUnexpectedLink		:=	inState.11;

SyncUnitHasSomeIssue :=	_state.AtLeastOneSlaveInInitState OR
						_state.AtLeastOneSlaveInPreopState OR
						_state.AtLeastOneSlaveInBootState OR
						_state.AtLeastOneSlaveInSafeOpState OR
						_state.AtLeastOneSlaveSignalsError OR
						_state.InvalidVendoridOrProductcodeRead OR
						_state.InitializationErrorOccurred OR
						_state.AtLeastOneSlaveNotPresent OR
						_state.AtLeastOneSlaveSignalsLinkError OR
						_state.AtLeastOneSlaveSignalsMissingLink OR
						_state.AtLeastOneSlaveSignalsUnexpectedLink;
END_METHOD

METHOD UpdateSyncUnitsStatus
VAR_INPUT
	SyncUnits			:	POINTER TO SyncUnitTask_B4157F22;
	SyncUnitsSize		:	UINT;
END_VAR
VAR
    _i					:	UINT;
	_pSyncUnit			:	POINTER TO SyncUnitTask_B4157F22;
	_SyncUnit			:	SyncUnitTask_B4157F22;
	_SyncUnitState		:	UINT;
END_VAR
_someSyncUnitHasSomeIssue := FALSE;
_allDataValid := TRUE;
_someDataInvalid := FALSE;

IF SyncUnits<>0 THEN
	_numberOfSyncUnits := SyncUnitsSize / SIZEOF(SyncUnitTask_B4157F22);
	FOR _i := 0 TO _numberOfSyncUnits - 1 DO
		_pSyncUnit					:=	SyncUnits + _i * SIZEOF(SyncUnitTask_B4157F22);
		_SyncUnit					:=	_pSyncUnit^;	
		_someSyncUnitHasSomeIssue 	:=	_someSyncUnitHasSomeIssue OR SyncUnitHasSomeIssue(_SyncUnit.InfoData.State);
		_allDataValid				:=	_allDataValid AND NOT _SyncUnit.WcState.WcState;
		_someDataInvalid			:=	_someDataInvalid OR _SyncUnit.WcState.WcState;
	END_FOR
END_IF
END_METHOD

END_FUNCTION_BLOCK

// ---- Diagnostics/EtherCAT/SyncUnit/TcoSyncUnit.TcPOU
FUNCTION_BLOCK TcoSyncUnit EXTENDS TcoCore.TcoObject IMPLEMENTS ITcoSyncUnit
VAR
    {attribute addProperty Name "WcState"}
    WcState : WcState_0B2B16F9;
    {attribute addProperty Name "InfoData"}
    InfoData : InfoData_2A97D6CF;
    {attribute addProperty Name "Status"}
    _State : SyncUnitState;
    {attribute 'hide'}
    _hasSomeIssue : BOOL;
    {attribute 'hide'}
    _dataValid : BOOL;
    {attribute 'hide'}
    _dataInvalid : BOOL;
END_VAR

PROPERTY DataInvalid : BOOL
GET
_dataInvalid := WcState.WcState;
DataInvalid := _dataInvalid;
END_GET
END_PROPERTY

PROPERTY DataValid : BOOL
GET
_dataValid := NOT WcState.WcState;
DataValid := _dataValid;
END_GET
END_PROPERTY

PROPERTY HasSomeIssue : BOOL
GET
VAR
	_syncUnitStatus : SyncUnitState;
END_VAR
_syncUnitStatus := State;

_hasSomeIssue := _syncUnitStatus.AtLeastOneSlaveInInitState OR
			_syncUnitStatus.AtLeastOneSlaveInPreopState OR
			_syncUnitStatus.AtLeastOneSlaveInBootState OR
			_syncUnitStatus.AtLeastOneSlaveInSafeOpState OR
			_syncUnitStatus.AtLeastOneSlaveSignalsError OR
			_syncUnitStatus.InvalidVendoridOrProductcodeRead OR
			_syncUnitStatus.InitializationErrorOccurred OR
			_syncUnitStatus.AtLeastOneSlaveNotPresent OR
			_syncUnitStatus.AtLeastOneSlaveSignalsLinkError OR
			_syncUnitStatus.AtLeastOneSlaveSignalsMissingLink OR
			_syncUnitStatus.AtLeastOneSlaveSignalsUnexpectedLink;
	
HasSomeIssue := _hasSomeIssue;
END_GET
END_PROPERTY

PROPERTY State : SyncUnitState
GET
_State.AtLeastOneSlaveInInitState := InfoData.State.0 AND NOT InfoData.State.1;
_State.AtLeastOneSlaveInPreopState := InfoData.State.0 AND InfoData.State.1;
_State.AtLeastOneSlaveInBootState := InfoData.State.0 AND InfoData.State.1;
_State.AtLeastOneSlaveInSafeOpState := InfoData.State.2;
_State.AtLeastOneSlaveInOpState := InfoData.State.3;
_State.AtLeastOneSlaveSignalsError := InfoData.State.4;
_State.InvalidVendoridOrProductcodeRead := InfoData.State.5;
_State.InitializationErrorOccurred := InfoData.State.6;
_State.AtLeastOneSlaveDisabled := InfoData.State.7;
_State.AtLeastOneSlaveNotPresent := InfoData.State.8;
_State.AtLeastOneSlaveSignalsLinkError := InfoData.State.9;
_State.AtLeastOneSlaveSignalsMissingLink := InfoData.State.10;
_State.AtLeastOneSlaveSignalsUnexpectedLink := InfoData.State.11;

State := _State;
END_GET
END_PROPERTY

END_FUNCTION_BLOCK

// ---- POUs/MAIN.TcPOU
PROGRAM MAIN
VAR
END_VAR

END_PROGRAM
